% RSLogix 500 project Planer 3-1-07.RSS, saved by version 7.00.00.19 %
PROJECT "PLANER"    % processor: MicroLogix 1500 %

PROGRAM FILES
  LAD 2 "MAIN"  13 rungs
  LAD 3 "INFEED"  10 rungs
  LAD 4 "TILTHOIST"  9 rungs
  LAD 5 "GRADING"  22 rungs
  LAD 6 "PLANER IF"  6 rungs
  LAD 7 "PLANER OF"  5 rungs
  LAD 8 "MR CONVS"  7 rungs
  LAD 9 "CYCLONE"  3 rungs
  LAD 10 "INDICATION"  11 rungs

DATA FILES
  O0 OUTPUT  9 elements
  I1 INPUT  8 elements
  S2 STATUS  66 elements
  B3 BINARY  10 elements
  T4 TIMER  34 elements
  C5 COUNTER  1 elements
  R6 CONTROL  1 elements
  N7 INTEGER  1 elements
  F8 FLOAT  1 elements

LADDER 2 "MAIN"
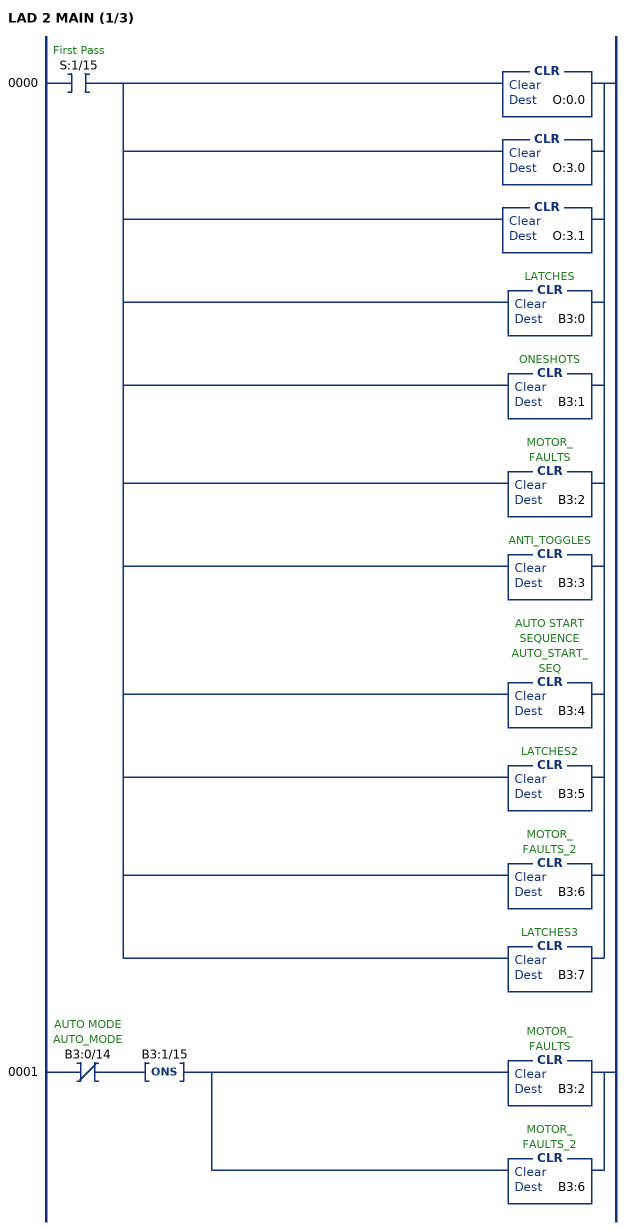
% Rung: 0 %
SOR XIC S:1/15 BST CLR O:0.0 NXB CLR O:3.0 NXB CLR O:3.1 NXB CLR B3:0 NXB CLR B3:1 NXB CLR B3:2 NXB CLR B3:3 NXB CLR B3:4 NXB CLR B3:5 NXB CLR B3:6 NXB CLR B3:7 BND EOR
%   S:1/15  "First Pass" %
%   B3:0  LATCHES %
%   B3:1  ONESHOTS %
%   B3:2  MOTOR_FAULTS %
%   B3:3  ANTI_TOGGLES %
%   B3:4  AUTO_START_SEQ  "AUTO START SEQUENCE" %
%   B3:5  LATCHES2 %
%   B3:6  MOTOR_FAULTS_2 %
%   B3:7  LATCHES3 %
% Rung: 1 %
SOR XIO B3:0/14 ONS B3:1/15 BST CLR B3:2 NXB CLR B3:6 BND EOR
%   B3:0/14  AUTO_MODE  "AUTO MODE" %
%   B3:2  MOTOR_FAULTS %
%   B3:6  MOTOR_FAULTS_2 %

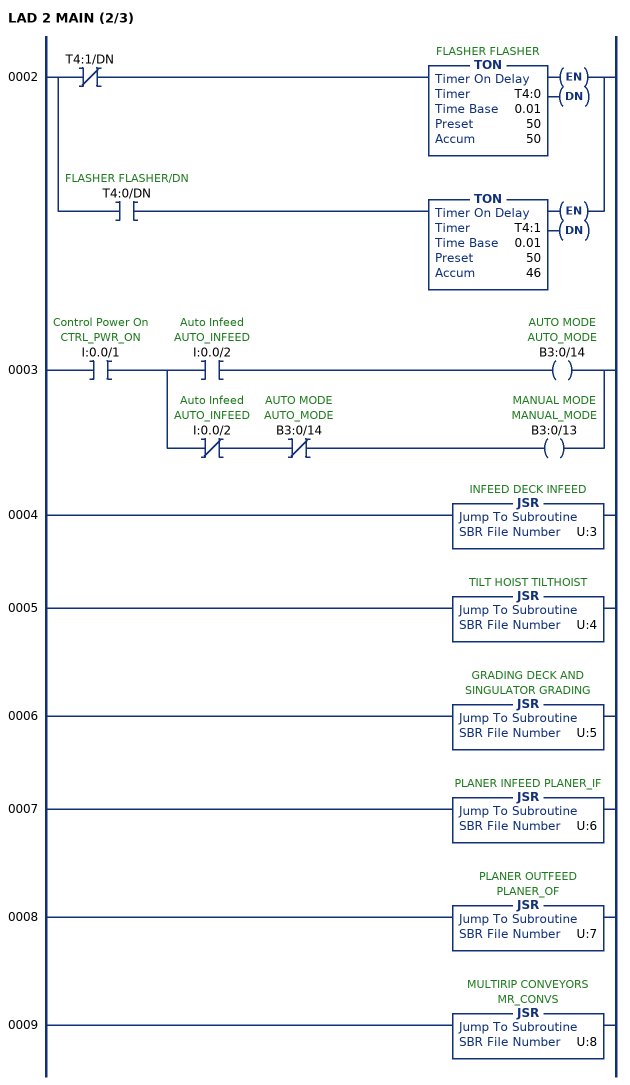
% Rung: 2 %
SOR BST XIO T4:1/DN TON T4:0 0.01 50 50 NXB XIC T4:0/DN TON T4:1 0.01 50 46 BND EOR
%   T4:0  FLASHER  "FLASHER" %
% Rung: 3 %
SOR XIC I:0.0/1 BST XIC I:0.0/2 OTE B3:0/14 NXB XIO I:0.0/2 XIO B3:0/14 OTE B3:0/13 BND EOR
%   I:0.0/1  CTRL_PWR_ON  "Control Power On" %
%   I:0.0/2  AUTO_INFEED  "Auto Infeed" %
%   B3:0/14  AUTO_MODE  "AUTO MODE" %
%   B3:0/13  MANUAL_MODE  "MANUAL MODE" %
% Rung: 4 %
SOR JSR U:3 EOR
%   U:3  INFEED  "INFEED DECK" %
% Rung: 5 %
SOR JSR U:4 EOR
%   U:4  TILTHOIST  "TILT HOIST" %
% Rung: 6 %
SOR JSR U:5 EOR
%   U:5  GRADING  "GRADING DECK AND SINGULATOR" %
% Rung: 7 %
SOR JSR U:6 EOR
%   U:6  PLANER_IF  "PLANER INFEED" %
% Rung: 8 %
SOR JSR U:7 EOR
%   U:7  PLANER_OF  "PLANER OUTFEED" %
% Rung: 9 %
SOR JSR U:8 EOR
%   U:8  MR_CONVS  "MULTIRIP CONVEYORS" %

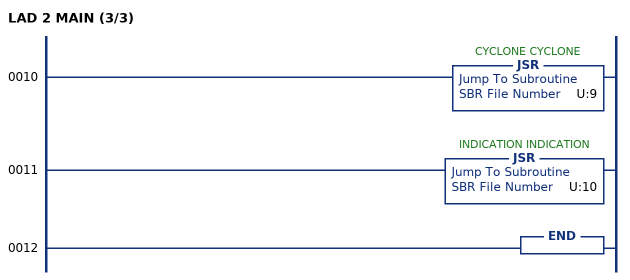
% Rung: 10 %
SOR JSR U:9 EOR
%   U:9  CYCLONE  "CYCLONE" %
% Rung: 11 %
SOR JSR U:10 EOR
%   U:10  INDICATION  "INDICATION" %
% Rung: 12 %
SOR END EOR

LADDER 3 "INFEED"
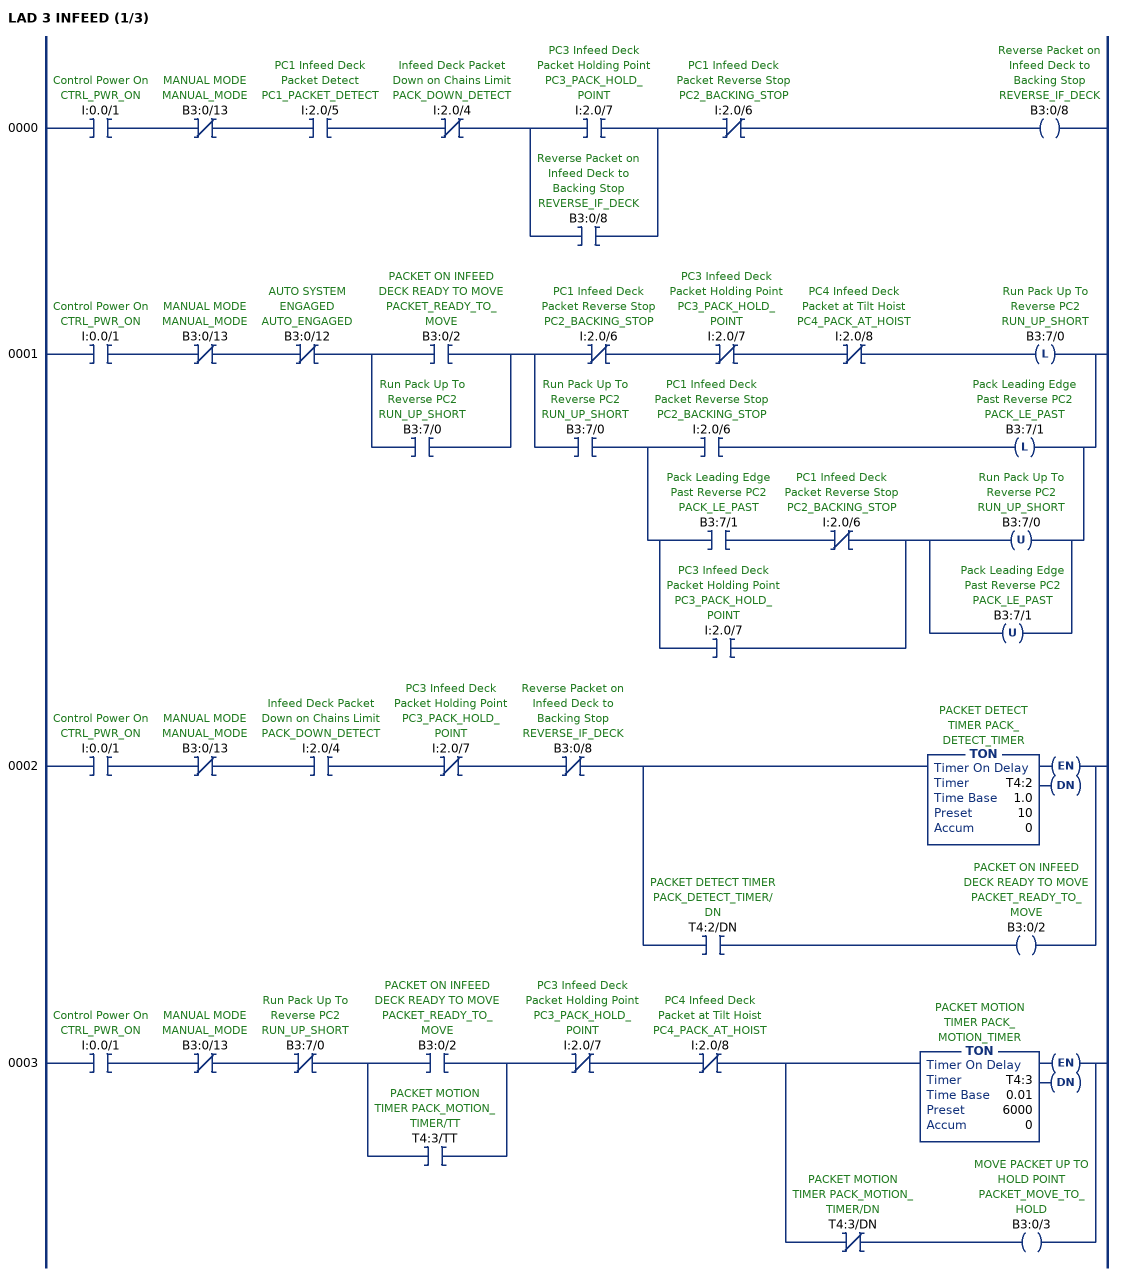
% Rung: 0 %
SOR XIC I:0.0/1 XIO B3:0/13 XIC I:2.0/5 XIO I:2.0/4 BST XIC I:2.0/7 NXB XIC B3:0/8 BND XIO I:2.0/6 OTE B3:0/8 EOR
%   I:0.0/1  CTRL_PWR_ON  "Control Power On" %
%   B3:0/13  MANUAL_MODE  "MANUAL MODE" %
%   I:2.0/5  PC1_PACKET_DETECT  "PC1 Infeed Deck Packet Detect" %
%   I:2.0/4  PACK_DOWN_DETECT  "Infeed Deck Packet Down on Chains Limit" %
%   I:2.0/7  PC3_PACK_HOLD_POINT  "PC3 Infeed Deck Packet Holding Point" %
%   B3:0/8  REVERSE_IF_DECK  "Reverse Packet on Infeed Deck to Backing Stop" %
%   I:2.0/6  PC2_BACKING_STOP  "PC1 Infeed Deck Packet Reverse Stop" %
% Rung: 1 %
SOR XIC I:0.0/1 XIO B3:0/13 XIO B3:0/12 BST XIC B3:0/2 NXB XIC B3:7/0 BND BST XIO I:2.0/6 XIO I:2.0/7 XIO I:2.0/8 OTL B3:7/0 NXB XIC B3:7/0 BST XIC I:2.0/6 OTL B3:7/1 NXB BST XIC B3:7/1 XIO I:2.0/6 NXB XIC I:2.0/7 BND BST OTU B3:7/0 NXB OTU B3:7/1 BND BND BND EOR
%   I:0.0/1  CTRL_PWR_ON  "Control Power On" %
%   B3:0/13  MANUAL_MODE  "MANUAL MODE" %
%   B3:0/12  AUTO_ENGAGED  "AUTO SYSTEM ENGAGED" %
%   B3:0/2  PACKET_READY_TO_MOVE  "PACKET ON INFEED DECK READY TO MOVE" %
%   B3:7/0  RUN_UP_SHORT  "Run Pack Up To Reverse PC2" %
%   I:2.0/6  PC2_BACKING_STOP  "PC1 Infeed Deck Packet Reverse Stop" %
%   I:2.0/7  PC3_PACK_HOLD_POINT  "PC3 Infeed Deck Packet Holding Point" %
%   I:2.0/8  PC4_PACK_AT_HOIST  "PC4 Infeed Deck Packet at Tilt Hoist" %
%   B3:7/1  PACK_LE_PAST  "Pack Leading Edge Past Reverse PC2" %
% Rung: 2 %
SOR XIC I:0.0/1 XIO B3:0/13 XIC I:2.0/4 XIO I:2.0/7 XIO B3:0/8 BST TON T4:2 1.0 10 0 NXB XIC T4:2/DN OTE B3:0/2 BND EOR
%   I:0.0/1  CTRL_PWR_ON  "Control Power On" %
%   B3:0/13  MANUAL_MODE  "MANUAL MODE" %
%   I:2.0/4  PACK_DOWN_DETECT  "Infeed Deck Packet Down on Chains Limit" %
%   I:2.0/7  PC3_PACK_HOLD_POINT  "PC3 Infeed Deck Packet Holding Point" %
%   B3:0/8  REVERSE_IF_DECK  "Reverse Packet on Infeed Deck to Backing Stop" %
%   T4:2  PACK_DETECT_TIMER  "PACKET DETECT TIMER" %
%   B3:0/2  PACKET_READY_TO_MOVE  "PACKET ON INFEED DECK READY TO MOVE" %
% Rung: 3 %
SOR XIC I:0.0/1 XIO B3:0/13 XIO B3:7/0 BST XIC B3:0/2 NXB XIC T4:3/TT BND XIO I:2.0/7 XIO I:2.0/8 BST TON T4:3 0.01 6000 0 NXB XIO T4:3/DN OTE B3:0/3 BND EOR
%   I:0.0/1  CTRL_PWR_ON  "Control Power On" %
%   B3:0/13  MANUAL_MODE  "MANUAL MODE" %
%   B3:7/0  RUN_UP_SHORT  "Run Pack Up To Reverse PC2" %
%   B3:0/2  PACKET_READY_TO_MOVE  "PACKET ON INFEED DECK READY TO MOVE" %
%   T4:3  PACK_MOTION_TIMER  "PACKET MOTION TIMER" %
%   I:2.0/7  PC3_PACK_HOLD_POINT  "PC3 Infeed Deck Packet Holding Point" %
%   I:2.0/8  PC4_PACK_AT_HOIST  "PC4 Infeed Deck Packet at Tilt Hoist" %
%   B3:0/3  PACKET_MOVE_TO_HOLD  "MOVE PACKET UP TO HOLD POINT" %

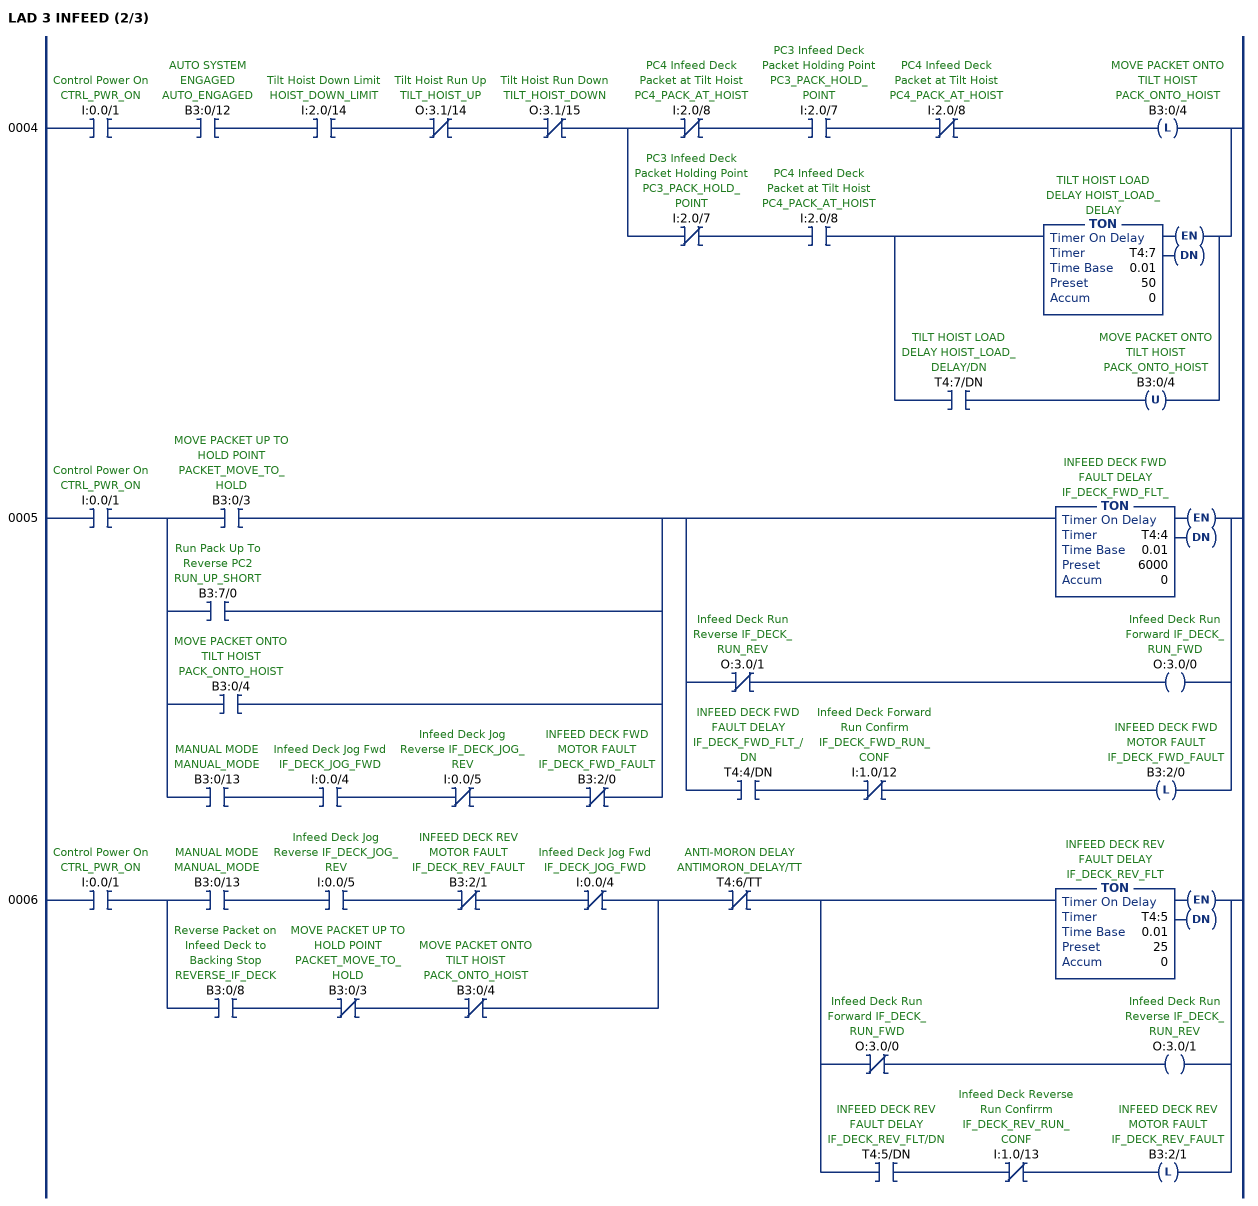
% Rung: 4 %
SOR XIC I:0.0/1 XIC B3:0/12 XIC I:2.0/14 XIO O:3.1/14 XIO O:3.1/15 BST XIO I:2.0/8 XIC I:2.0/7 XIO I:2.0/8 OTL B3:0/4 NXB XIO I:2.0/7 XIC I:2.0/8 BST TON T4:7 0.01 50 0 NXB XIC T4:7/DN OTU B3:0/4 BND BND EOR
%   I:0.0/1  CTRL_PWR_ON  "Control Power On" %
%   B3:0/12  AUTO_ENGAGED  "AUTO SYSTEM ENGAGED" %
%   I:2.0/14  HOIST_DOWN_LIMIT  "Tilt Hoist Down Limit" %
%   O:3.1/14  TILT_HOIST_UP  "Tilt Hoist Run Up" %
%   O:3.1/15  TILT_HOIST_DOWN  "Tilt Hoist Run Down" %
%   I:2.0/8  PC4_PACK_AT_HOIST  "PC4 Infeed Deck Packet at Tilt Hoist" %
%   I:2.0/7  PC3_PACK_HOLD_POINT  "PC3 Infeed Deck Packet Holding Point" %
%   B3:0/4  PACK_ONTO_HOIST  "MOVE PACKET ONTO TILT HOIST" %
%   T4:7  HOIST_LOAD_DELAY  "TILT HOIST LOAD DELAY" %
% Rung: 5 %
SOR XIC I:0.0/1 BST BST XIC B3:0/3 NXB XIC B3:7/0 NXB XIC B3:0/4 BND NXB XIC B3:0/13 XIC I:0.0/4 XIO I:0.0/5 XIO B3:2/0 BND BST TON T4:4 0.01 6000 0 NXB XIO O:3.0/1 OTE O:3.0/0 NXB XIC T4:4/DN XIO I:1.0/12 OTL B3:2/0 BND EOR
%   I:0.0/1  CTRL_PWR_ON  "Control Power On" %
%   B3:0/3  PACKET_MOVE_TO_HOLD  "MOVE PACKET UP TO HOLD POINT" %
%   B3:7/0  RUN_UP_SHORT  "Run Pack Up To Reverse PC2" %
%   B3:0/4  PACK_ONTO_HOIST  "MOVE PACKET ONTO TILT HOIST" %
%   B3:0/13  MANUAL_MODE  "MANUAL MODE" %
%   I:0.0/4  IF_DECK_JOG_FWD  "Infeed Deck Jog Fwd" %
%   I:0.0/5  IF_DECK_JOG_REV  "Infeed Deck Jog Reverse" %
%   B3:2/0  IF_DECK_FWD_FAULT  "INFEED DECK FWD MOTOR FAULT" %
%   T4:4  IF_DECK_FWD_FLT_  "INFEED DECK FWD FAULT DELAY" %
%   O:3.0/1  IF_DECK_RUN_REV  "Infeed Deck Run Reverse" %
%   O:3.0/0  IF_DECK_RUN_FWD  "Infeed Deck Run Forward" %
%   I:1.0/12  IF_DECK_FWD_RUN_CONF  "Infeed Deck Forward Run Confirm" %
% Rung: 6 %
SOR XIC I:0.0/1 BST XIC B3:0/13 XIC I:0.0/5 XIO B3:2/1 XIO I:0.0/4 NXB XIC B3:0/8 XIO B3:0/3 XIO B3:0/4 BND XIO T4:6/TT BST TON T4:5 0.01 25 0 NXB XIO O:3.0/0 OTE O:3.0/1 NXB XIC T4:5/DN XIO I:1.0/13 OTL B3:2/1 BND EOR
%   I:0.0/1  CTRL_PWR_ON  "Control Power On" %
%   B3:0/13  MANUAL_MODE  "MANUAL MODE" %
%   I:0.0/5  IF_DECK_JOG_REV  "Infeed Deck Jog Reverse" %
%   B3:2/1  IF_DECK_REV_FAULT  "INFEED DECK REV MOTOR FAULT" %
%   I:0.0/4  IF_DECK_JOG_FWD  "Infeed Deck Jog Fwd" %
%   B3:0/8  REVERSE_IF_DECK  "Reverse Packet on Infeed Deck to Backing Stop" %
%   B3:0/3  PACKET_MOVE_TO_HOLD  "MOVE PACKET UP TO HOLD POINT" %
%   B3:0/4  PACK_ONTO_HOIST  "MOVE PACKET ONTO TILT HOIST" %
%   T4:6  ANTIMORON_DELAY  "ANTI-MORON DELAY" %
%   T4:5  IF_DECK_REV_FLT  "INFEED DECK REV FAULT DELAY" %
%   O:3.0/0  IF_DECK_RUN_FWD  "Infeed Deck Run Forward" %
%   O:3.0/1  IF_DECK_RUN_REV  "Infeed Deck Run Reverse" %
%   I:1.0/13  IF_DECK_REV_RUN_CONF  "Infeed Deck Reverse Run Confirrm" %

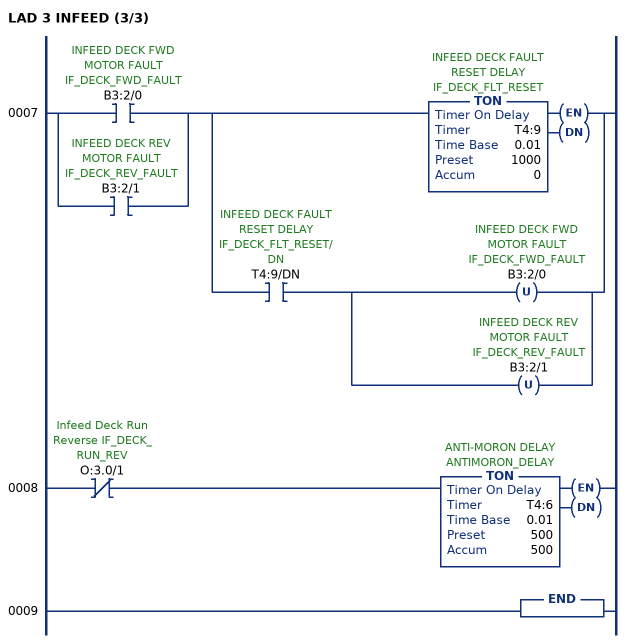
% Rung: 7 %
SOR BST XIC B3:2/0 NXB XIC B3:2/1 BND BST TON T4:9 0.01 1000 0 NXB XIC T4:9/DN BST OTU B3:2/0 NXB OTU B3:2/1 BND BND EOR
%   B3:2/0  IF_DECK_FWD_FAULT  "INFEED DECK FWD MOTOR FAULT" %
%   B3:2/1  IF_DECK_REV_FAULT  "INFEED DECK REV MOTOR FAULT" %
%   T4:9  IF_DECK_FLT_RESET  "INFEED DECK FAULT RESET DELAY" %
% Rung: 8 %
SOR XIO O:3.0/1 TON T4:6 0.01 500 500 EOR
%   O:3.0/1  IF_DECK_RUN_REV  "Infeed Deck Run Reverse" %
%   T4:6  ANTIMORON_DELAY  "ANTI-MORON DELAY" %
% Rung: 9 %
SOR END EOR

LADDER 4 "TILTHOIST"
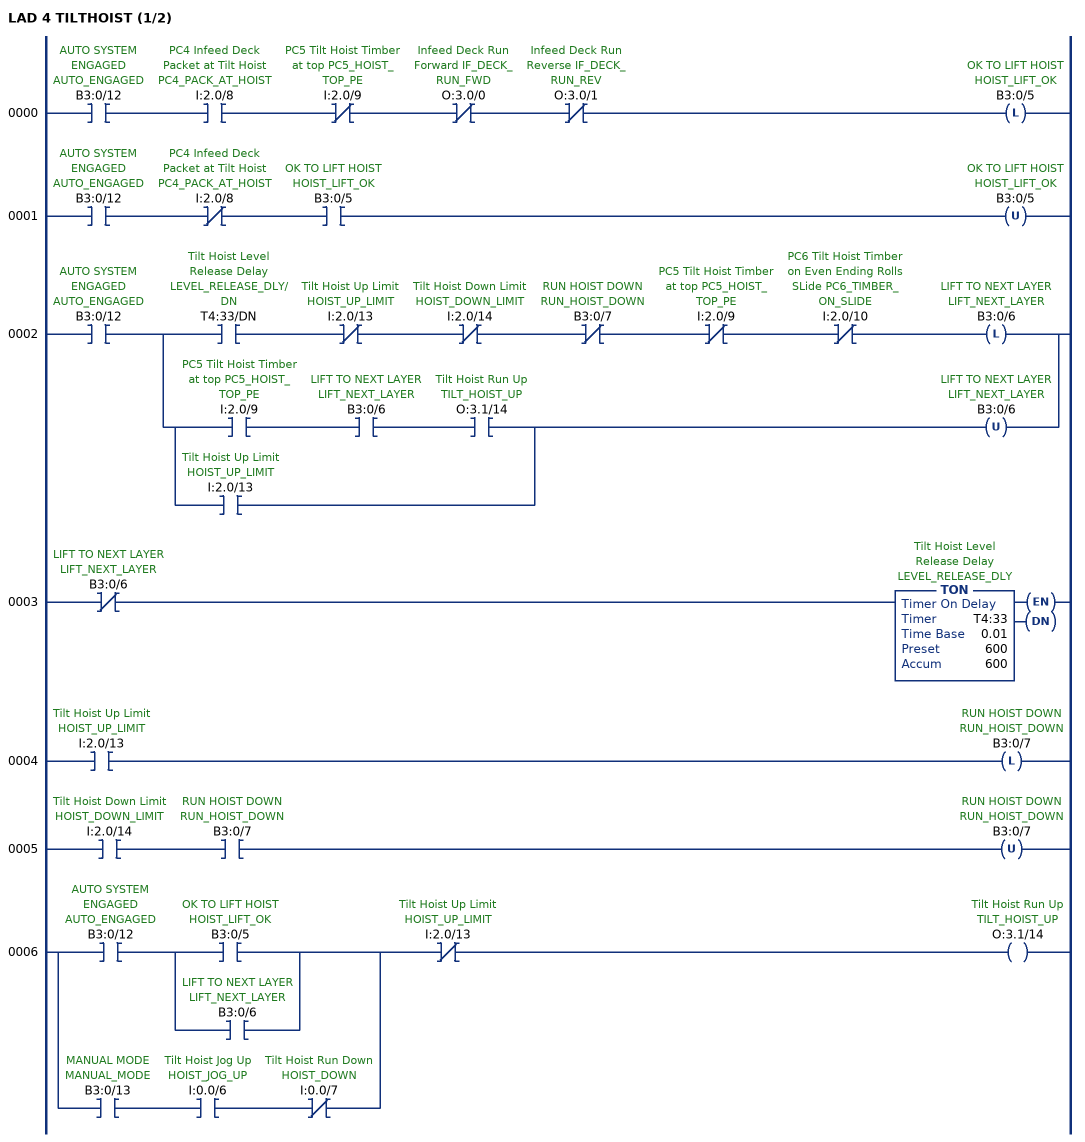
% Rung: 0 %
SOR XIC B3:0/12 XIC I:2.0/8 XIO I:2.0/9 XIO O:3.0/0 XIO O:3.0/1 OTL B3:0/5 EOR
%   B3:0/12  AUTO_ENGAGED  "AUTO SYSTEM ENGAGED" %
%   I:2.0/8  PC4_PACK_AT_HOIST  "PC4 Infeed Deck Packet at Tilt Hoist" %
%   I:2.0/9  PC5_HOIST_TOP_PE  "PC5 Tilt Hoist Timber at top" %
%   O:3.0/0  IF_DECK_RUN_FWD  "Infeed Deck Run Forward" %
%   O:3.0/1  IF_DECK_RUN_REV  "Infeed Deck Run Reverse" %
%   B3:0/5  HOIST_LIFT_OK  "OK TO LIFT HOIST" %
% Rung: 1 %
SOR XIC B3:0/12 XIO I:2.0/8 XIC B3:0/5 OTU B3:0/5 EOR
%   B3:0/12  AUTO_ENGAGED  "AUTO SYSTEM ENGAGED" %
%   I:2.0/8  PC4_PACK_AT_HOIST  "PC4 Infeed Deck Packet at Tilt Hoist" %
%   B3:0/5  HOIST_LIFT_OK  "OK TO LIFT HOIST" %
% Rung: 2 %
SOR XIC B3:0/12 BST XIC T4:33/DN XIO I:2.0/13 XIO I:2.0/14 XIO B3:0/7 XIO I:2.0/9 XIO I:2.0/10 OTL B3:0/6 NXB BST XIC I:2.0/9 XIC B3:0/6 XIC O:3.1/14 NXB XIC I:2.0/13 BND OTU B3:0/6 BND EOR
%   B3:0/12  AUTO_ENGAGED  "AUTO SYSTEM ENGAGED" %
%   T4:33  LEVEL_RELEASE_DLY  "Tilt Hoist Level Release Delay" %
%   I:2.0/13  HOIST_UP_LIMIT  "Tilt Hoist Up Limit" %
%   I:2.0/14  HOIST_DOWN_LIMIT  "Tilt Hoist Down Limit" %
%   B3:0/7  RUN_HOIST_DOWN  "RUN HOIST DOWN" %
%   I:2.0/9  PC5_HOIST_TOP_PE  "PC5 Tilt Hoist Timber at top" %
%   I:2.0/10  PC6_TIMBER_ON_SLIDE  "PC6 Tilt Hoist Timber on Even Ending Rolls SLide" %
%   B3:0/6  LIFT_NEXT_LAYER  "LIFT TO NEXT LAYER" %
%   O:3.1/14  TILT_HOIST_UP  "Tilt Hoist Run Up" %
% Rung: 3 %
SOR XIO B3:0/6 TON T4:33 0.01 600 600 EOR
%   B3:0/6  LIFT_NEXT_LAYER  "LIFT TO NEXT LAYER" %
%   T4:33  LEVEL_RELEASE_DLY  "Tilt Hoist Level Release Delay" %
% Rung: 4 %
SOR XIC I:2.0/13 OTL B3:0/7 EOR
%   I:2.0/13  HOIST_UP_LIMIT  "Tilt Hoist Up Limit" %
%   B3:0/7  RUN_HOIST_DOWN  "RUN HOIST DOWN" %
% Rung: 5 %
SOR XIC I:2.0/14 XIC B3:0/7 OTU B3:0/7 EOR
%   I:2.0/14  HOIST_DOWN_LIMIT  "Tilt Hoist Down Limit" %
%   B3:0/7  RUN_HOIST_DOWN  "RUN HOIST DOWN" %
% Rung: 6 %
SOR BST XIC B3:0/12 BST XIC B3:0/5 NXB XIC B3:0/6 BND NXB XIC B3:0/13 XIC I:0.0/6 XIO I:0.0/7 BND XIO I:2.0/13 OTE O:3.1/14 EOR
%   B3:0/12  AUTO_ENGAGED  "AUTO SYSTEM ENGAGED" %
%   B3:0/5  HOIST_LIFT_OK  "OK TO LIFT HOIST" %
%   B3:0/6  LIFT_NEXT_LAYER  "LIFT TO NEXT LAYER" %
%   B3:0/13  MANUAL_MODE  "MANUAL MODE" %
%   I:0.0/6  HOIST_JOG_UP  "Tilt Hoist Jog Up" %
%   I:0.0/7  HOIST_DOWN  "Tilt Hoist Run Down" %
%   I:2.0/13  HOIST_UP_LIMIT  "Tilt Hoist Up Limit" %
%   O:3.1/14  TILT_HOIST_UP  "Tilt Hoist Run Up" %

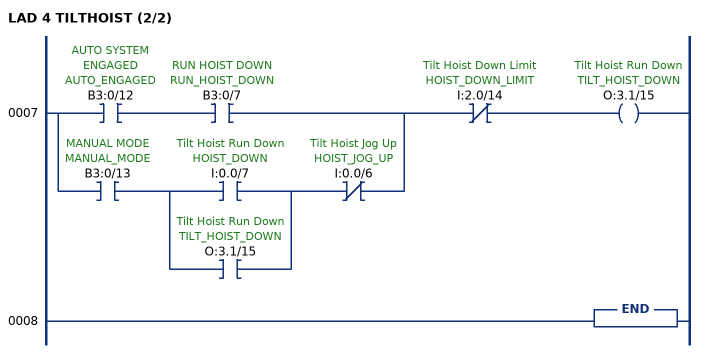
% Rung: 7 %
SOR BST XIC B3:0/12 XIC B3:0/7 NXB XIC B3:0/13 BST XIC I:0.0/7 NXB XIC O:3.1/15 BND XIO I:0.0/6 BND XIO I:2.0/14 OTE O:3.1/15 EOR
%   B3:0/12  AUTO_ENGAGED  "AUTO SYSTEM ENGAGED" %
%   B3:0/7  RUN_HOIST_DOWN  "RUN HOIST DOWN" %
%   B3:0/13  MANUAL_MODE  "MANUAL MODE" %
%   I:0.0/7  HOIST_DOWN  "Tilt Hoist Run Down" %
%   O:3.1/15  TILT_HOIST_DOWN  "Tilt Hoist Run Down" %
%   I:0.0/6  HOIST_JOG_UP  "Tilt Hoist Jog Up" %
%   I:2.0/14  HOIST_DOWN_LIMIT  "Tilt Hoist Down Limit" %
% Rung: 8 %
SOR END EOR

LADDER 5 "GRADING"
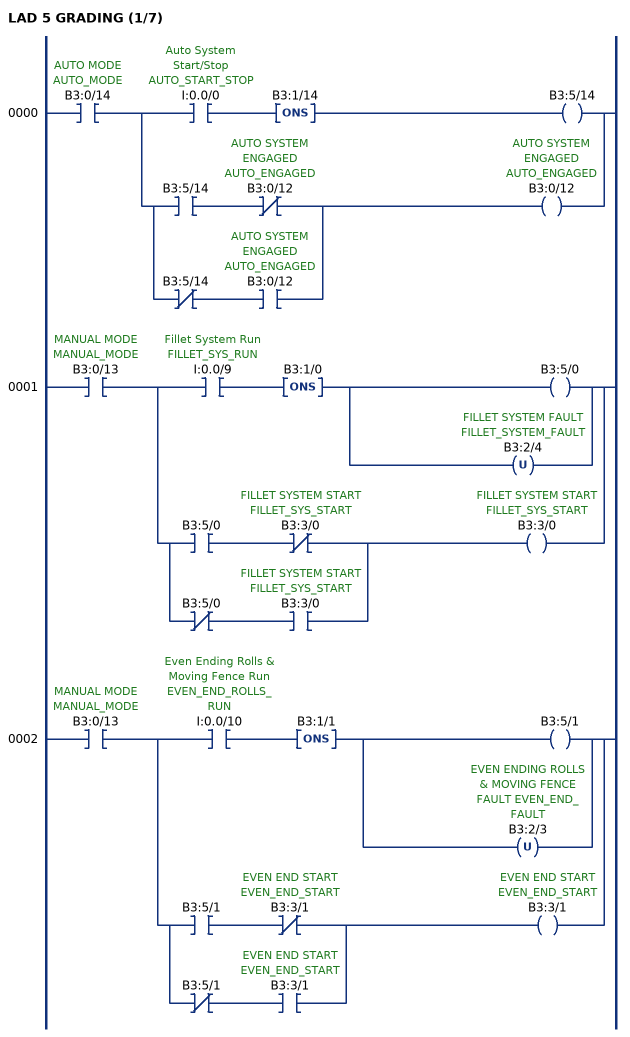
% Rung: 0 %
SOR XIC B3:0/14 BST XIC I:0.0/0 ONS B3:1/14 OTE B3:5/14 NXB BST XIC B3:5/14 XIO B3:0/12 NXB XIO B3:5/14 XIC B3:0/12 BND OTE B3:0/12 BND EOR
%   B3:0/14  AUTO_MODE  "AUTO MODE" %
%   I:0.0/0  AUTO_START_STOP  "Auto System Start/Stop" %
%   B3:0/12  AUTO_ENGAGED  "AUTO SYSTEM ENGAGED" %
% Rung: 1 %
SOR XIC B3:0/13 BST XIC I:0.0/9 ONS B3:1/0 BST OTE B3:5/0 NXB OTU B3:2/4 BND NXB BST XIC B3:5/0 XIO B3:3/0 NXB XIO B3:5/0 XIC B3:3/0 BND OTE B3:3/0 BND EOR
%   B3:0/13  MANUAL_MODE  "MANUAL MODE" %
%   I:0.0/9  FILLET_SYS_RUN  "Fillet System Run" %
%   B3:2/4  FILLET_SYSTEM_FAULT  "FILLET SYSTEM FAULT" %
%   B3:3/0  FILLET_SYS_START  "FILLET SYSTEM START" %
% Rung: 2 %
SOR XIC B3:0/13 BST XIC I:0.0/10 ONS B3:1/1 BST OTE B3:5/1 NXB OTU B3:2/3 BND NXB BST XIC B3:5/1 XIO B3:3/1 NXB XIO B3:5/1 XIC B3:3/1 BND OTE B3:3/1 BND EOR
%   B3:0/13  MANUAL_MODE  "MANUAL MODE" %
%   I:0.0/10  EVEN_END_ROLLS_RUN  "Even Ending Rolls & Moving Fence Run" %
%   B3:2/3  EVEN_END_FAULT  "EVEN ENDING ROLLS & MOVING FENCE FAULT" %
%   B3:3/1  EVEN_END_START  "EVEN END START" %

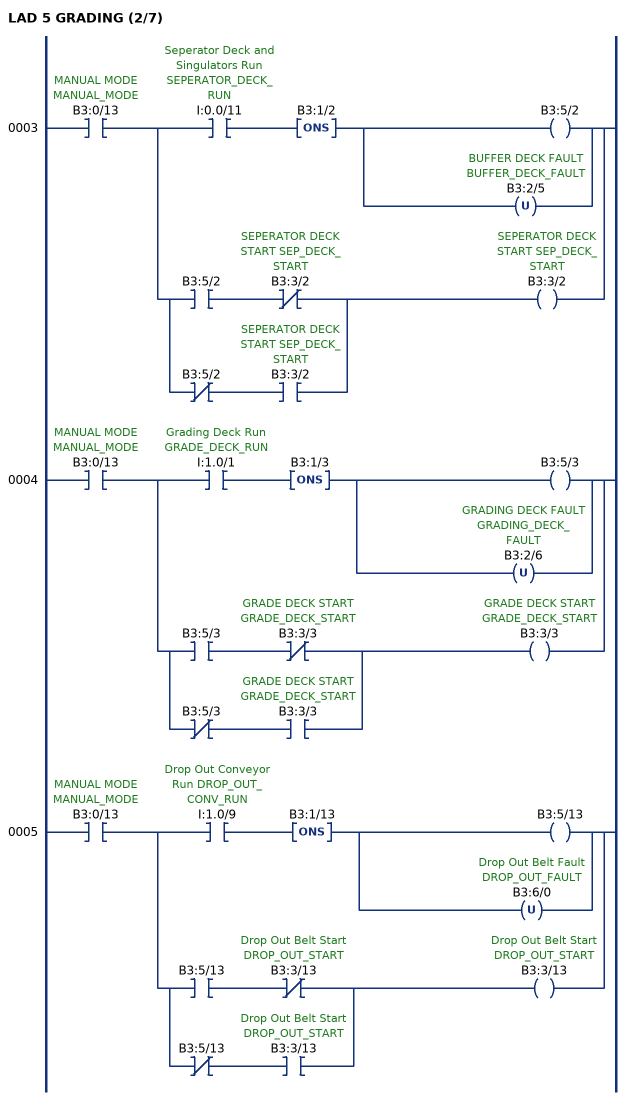
% Rung: 3 %
SOR XIC B3:0/13 BST XIC I:0.0/11 ONS B3:1/2 BST OTE B3:5/2 NXB OTU B3:2/5 BND NXB BST XIC B3:5/2 XIO B3:3/2 NXB XIO B3:5/2 XIC B3:3/2 BND OTE B3:3/2 BND EOR
%   B3:0/13  MANUAL_MODE  "MANUAL MODE" %
%   I:0.0/11  SEPERATOR_DECK_RUN  "Seperator Deck and Singulators Run" %
%   B3:2/5  BUFFER_DECK_FAULT  "BUFFER DECK FAULT" %
%   B3:3/2  SEP_DECK_START  "SEPERATOR DECK START" %
% Rung: 4 %
SOR XIC B3:0/13 BST XIC I:1.0/1 ONS B3:1/3 BST OTE B3:5/3 NXB OTU B3:2/6 BND NXB BST XIC B3:5/3 XIO B3:3/3 NXB XIO B3:5/3 XIC B3:3/3 BND OTE B3:3/3 BND EOR
%   B3:0/13  MANUAL_MODE  "MANUAL MODE" %
%   I:1.0/1  GRADE_DECK_RUN  "Grading Deck Run" %
%   B3:2/6  GRADING_DECK_FAULT  "GRADING DECK FAULT" %
%   B3:3/3  GRADE_DECK_START  "GRADE DECK START" %
% Rung: 5 %
SOR XIC B3:0/13 BST XIC I:1.0/9 ONS B3:1/13 BST OTE B3:5/13 NXB OTU B3:6/0 BND NXB BST XIC B3:5/13 XIO B3:3/13 NXB XIO B3:5/13 XIC B3:3/13 BND OTE B3:3/13 BND EOR
%   B3:0/13  MANUAL_MODE  "MANUAL MODE" %
%   I:1.0/9  DROP_OUT_CONV_RUN  "Drop Out Conveyor Run" %
%   B3:6/0  DROP_OUT_FAULT  "Drop Out Belt Fault" %
%   B3:3/13  DROP_OUT_START  "Drop Out Belt Start" %

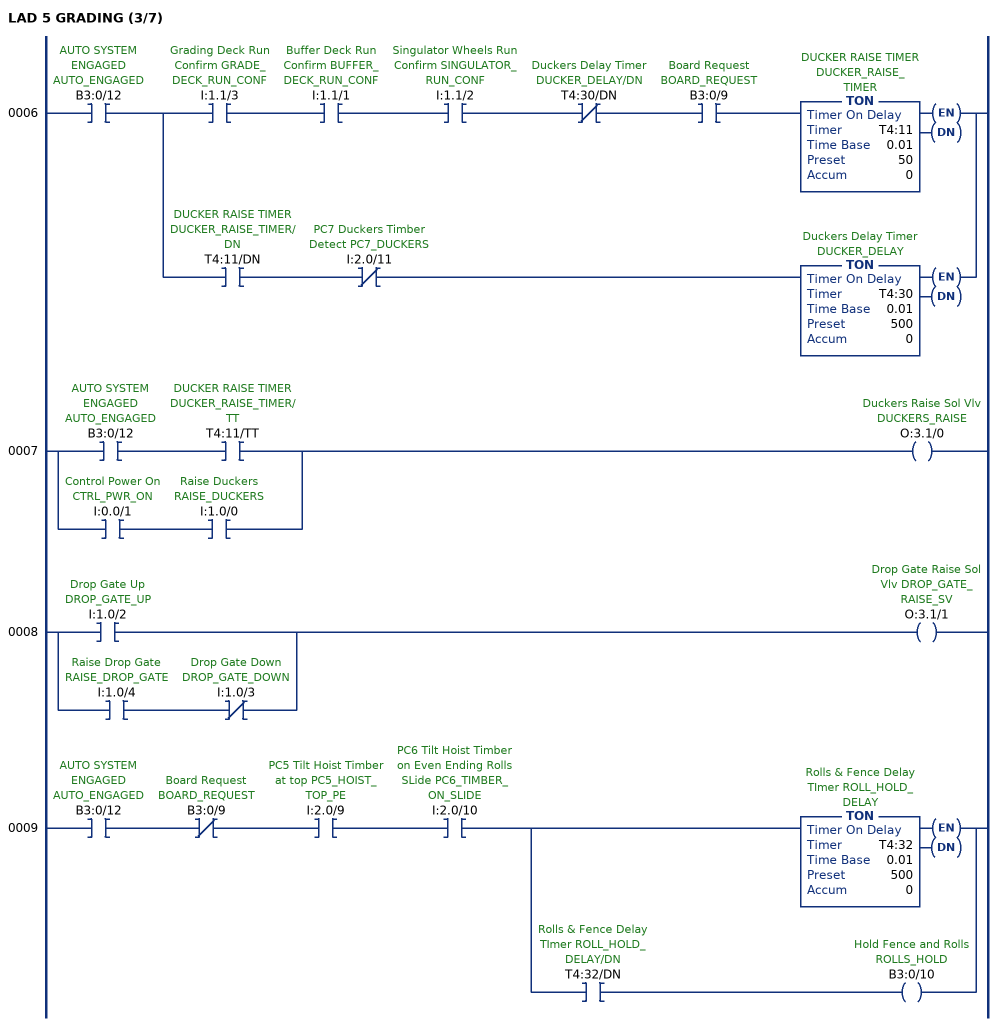
% Rung: 6 %
SOR XIC B3:0/12 BST XIC I:1.1/3 XIC I:1.1/1 XIC I:1.1/2 XIO T4:30/DN XIC B3:0/9 TON T4:11 0.01 50 0 NXB XIC T4:11/DN XIO I:2.0/11 TON T4:30 0.01 500 0 BND EOR
%   B3:0/12  AUTO_ENGAGED  "AUTO SYSTEM ENGAGED" %
%   I:1.1/3  GRADE_DECK_RUN_CONF  "Grading Deck Run Confirm" %
%   I:1.1/1  BUFFER_DECK_RUN_CONF  "Buffer Deck Run Confirm" %
%   I:1.1/2  SINGULATOR_RUN_CONF  "Singulator Wheels Run Confirm" %
%   T4:30  DUCKER_DELAY  "Duckers Delay Timer" %
%   B3:0/9  BOARD_REQUEST  "Board Request" %
%   T4:11  DUCKER_RAISE_TIMER  "DUCKER RAISE TIMER" %
%   I:2.0/11  PC7_DUCKERS  "PC7 Duckers Timber Detect" %
% Rung: 7 %
SOR BST XIC B3:0/12 XIC T4:11/TT NXB XIC I:0.0/1 XIC I:1.0/0 BND OTE O:3.1/0 EOR
%   B3:0/12  AUTO_ENGAGED  "AUTO SYSTEM ENGAGED" %
%   T4:11  DUCKER_RAISE_TIMER  "DUCKER RAISE TIMER" %
%   I:0.0/1  CTRL_PWR_ON  "Control Power On" %
%   I:1.0/0  RAISE_DUCKERS  "Raise Duckers" %
%   O:3.1/0  DUCKERS_RAISE  "Duckers Raise Sol Vlv" %
% Rung: 8 %
SOR BST XIC I:1.0/2 NXB XIC I:1.0/4 XIO I:1.0/3 BND OTE O:3.1/1 EOR
%   I:1.0/2  DROP_GATE_UP  "Drop Gate Up" %
%   I:1.0/4  RAISE_DROP_GATE  "Raise Drop Gate" %
%   I:1.0/3  DROP_GATE_DOWN  "Drop Gate Down" %
%   O:3.1/1  DROP_GATE_RAISE_SV  "Drop Gate Raise Sol Vlv" %
% Rung: 9 %
SOR XIC B3:0/12 XIO B3:0/9 XIC I:2.0/9 XIC I:2.0/10 BST TON T4:32 0.01 500 0 NXB XIC T4:32/DN OTE B3:0/10 BND EOR
%   B3:0/12  AUTO_ENGAGED  "AUTO SYSTEM ENGAGED" %
%   B3:0/9  BOARD_REQUEST  "Board Request" %
%   I:2.0/9  PC5_HOIST_TOP_PE  "PC5 Tilt Hoist Timber at top" %
%   I:2.0/10  PC6_TIMBER_ON_SLIDE  "PC6 Tilt Hoist Timber on Even Ending Rolls SLide" %
%   T4:32  ROLL_HOLD_DELAY  "Rolls & Fence Delay TImer" %
%   B3:0/10  ROLLS_HOLD  "Hold Fence and Rolls" %

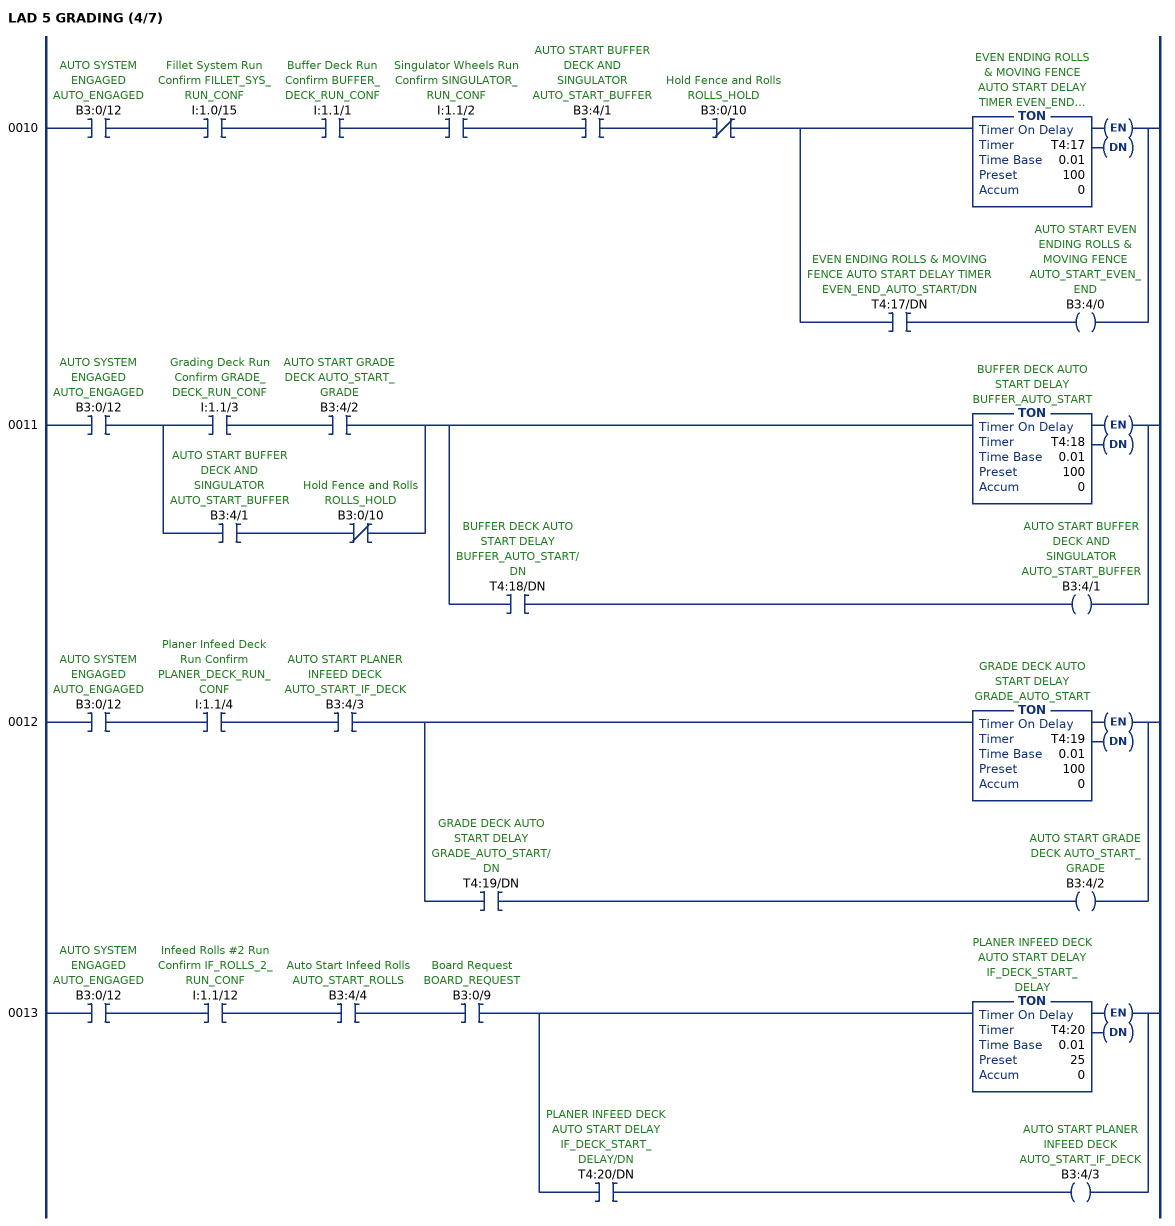
% Rung: 10 %
SOR XIC B3:0/12 XIC I:1.0/15 XIC I:1.1/1 XIC I:1.1/2 XIC B3:4/1 XIO B3:0/10 BST TON T4:17 0.01 100 0 NXB XIC T4:17/DN OTE B3:4/0 BND EOR
%   B3:0/12  AUTO_ENGAGED  "AUTO SYSTEM ENGAGED" %
%   I:1.0/15  FILLET_SYS_RUN_CONF  "Fillet System Run Confirm" %
%   I:1.1/1  BUFFER_DECK_RUN_CONF  "Buffer Deck Run Confirm" %
%   I:1.1/2  SINGULATOR_RUN_CONF  "Singulator Wheels Run Confirm" %
%   B3:4/1  AUTO_START_BUFFER  "AUTO START BUFFER DECK AND SINGULATOR" %
%   B3:0/10  ROLLS_HOLD  "Hold Fence and Rolls" %
%   T4:17  EVEN_END_AUTO_START  "EVEN ENDING ROLLS & MOVING FENCE AUTO START DELAY TIMER" %
%   B3:4/0  AUTO_START_EVEN_END  "AUTO START EVEN ENDING ROLLS & MOVING FENCE" %
% Rung: 11 %
SOR XIC B3:0/12 BST XIC I:1.1/3 XIC B3:4/2 NXB XIC B3:4/1 XIO B3:0/10 BND BST TON T4:18 0.01 100 0 NXB XIC T4:18/DN OTE B3:4/1 BND EOR
%   B3:0/12  AUTO_ENGAGED  "AUTO SYSTEM ENGAGED" %
%   I:1.1/3  GRADE_DECK_RUN_CONF  "Grading Deck Run Confirm" %
%   B3:4/2  AUTO_START_GRADE  "AUTO START GRADE DECK" %
%   B3:4/1  AUTO_START_BUFFER  "AUTO START BUFFER DECK AND SINGULATOR" %
%   B3:0/10  ROLLS_HOLD  "Hold Fence and Rolls" %
%   T4:18  BUFFER_AUTO_START  "BUFFER DECK AUTO START DELAY" %
% Rung: 12 %
SOR XIC B3:0/12 XIC I:1.1/4 XIC B3:4/3 BST TON T4:19 0.01 100 0 NXB XIC T4:19/DN OTE B3:4/2 BND EOR
%   B3:0/12  AUTO_ENGAGED  "AUTO SYSTEM ENGAGED" %
%   I:1.1/4  PLANER_DECK_RUN_CONF  "Planer Infeed Deck Run Confirm" %
%   B3:4/3  AUTO_START_IF_DECK  "AUTO START PLANER INFEED DECK" %
%   T4:19  GRADE_AUTO_START  "GRADE DECK AUTO START DELAY" %
%   B3:4/2  AUTO_START_GRADE  "AUTO START GRADE DECK" %
% Rung: 13 %
SOR XIC B3:0/12 XIC I:1.1/12 XIC B3:4/4 XIC B3:0/9 BST TON T4:20 0.01 25 0 NXB XIC T4:20/DN OTE B3:4/3 BND EOR
%   B3:0/12  AUTO_ENGAGED  "AUTO SYSTEM ENGAGED" %
%   I:1.1/12  IF_ROLLS_2_RUN_CONF  "Infeed Rolls #2 Run Confirm" %
%   B3:4/4  AUTO_START_ROLLS  "Auto Start Infeed Rolls" %
%   B3:0/9  BOARD_REQUEST  "Board Request" %
%   T4:20  IF_DECK_START_DELAY  "PLANER INFEED DECK AUTO START DELAY" %
%   B3:4/3  AUTO_START_IF_DECK  "AUTO START PLANER INFEED DECK" %

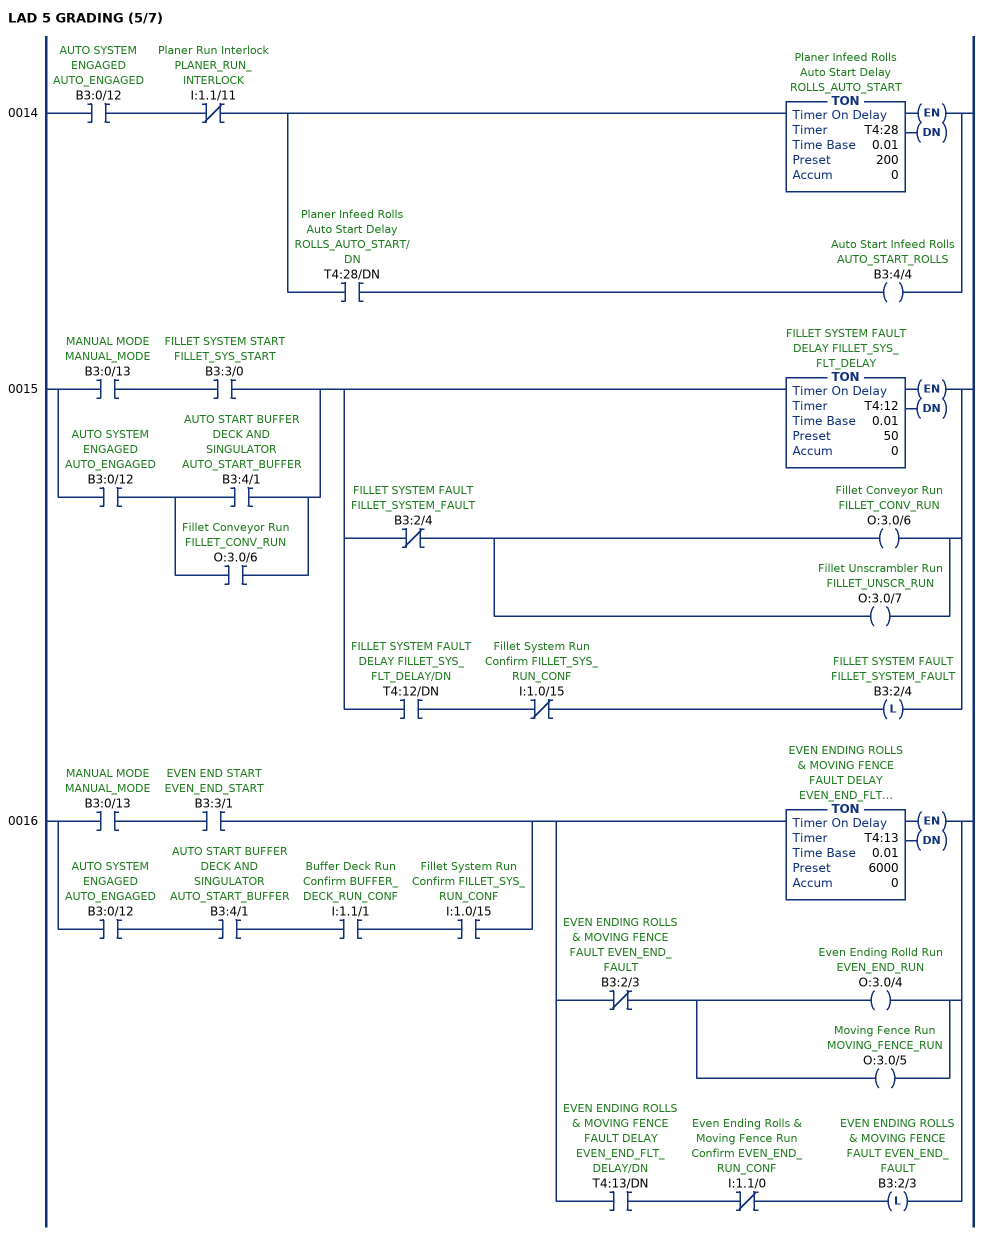
% Rung: 14 %
SOR XIC B3:0/12 XIO I:1.1/11 BST TON T4:28 0.01 200 0 NXB XIC T4:28/DN OTE B3:4/4 BND EOR
%   B3:0/12  AUTO_ENGAGED  "AUTO SYSTEM ENGAGED" %
%   I:1.1/11  PLANER_RUN_INTERLOCK  "Planer Run Interlock" %
%   T4:28  ROLLS_AUTO_START  "Planer Infeed Rolls Auto Start Delay" %
%   B3:4/4  AUTO_START_ROLLS  "Auto Start Infeed Rolls" %
% Rung: 15 %
SOR BST XIC B3:0/13 XIC B3:3/0 NXB XIC B3:0/12 BST XIC B3:4/1 NXB XIC O:3.0/6 BND BND BST TON T4:12 0.01 50 0 NXB XIO B3:2/4 BST OTE O:3.0/6 NXB OTE O:3.0/7 BND NXB XIC T4:12/DN XIO I:1.0/15 OTL B3:2/4 BND EOR
%   B3:0/13  MANUAL_MODE  "MANUAL MODE" %
%   B3:3/0  FILLET_SYS_START  "FILLET SYSTEM START" %
%   B3:0/12  AUTO_ENGAGED  "AUTO SYSTEM ENGAGED" %
%   B3:4/1  AUTO_START_BUFFER  "AUTO START BUFFER DECK AND SINGULATOR" %
%   O:3.0/6  FILLET_CONV_RUN  "Fillet Conveyor Run" %
%   T4:12  FILLET_SYS_FLT_DELAY  "FILLET SYSTEM FAULT DELAY" %
%   B3:2/4  FILLET_SYSTEM_FAULT  "FILLET SYSTEM FAULT" %
%   O:3.0/7  FILLET_UNSCR_RUN  "Fillet Unscrambler Run" %
%   I:1.0/15  FILLET_SYS_RUN_CONF  "Fillet System Run Confirm" %
% Rung: 16 %
SOR BST XIC B3:0/13 XIC B3:3/1 NXB XIC B3:0/12 XIC B3:4/1 XIC I:1.1/1 XIC I:1.0/15 BND BST TON T4:13 0.01 6000 0 NXB XIO B3:2/3 BST OTE O:3.0/4 NXB OTE O:3.0/5 BND NXB XIC T4:13/DN XIO I:1.1/0 OTL B3:2/3 BND EOR
%   B3:0/13  MANUAL_MODE  "MANUAL MODE" %
%   B3:3/1  EVEN_END_START  "EVEN END START" %
%   B3:0/12  AUTO_ENGAGED  "AUTO SYSTEM ENGAGED" %
%   B3:4/1  AUTO_START_BUFFER  "AUTO START BUFFER DECK AND SINGULATOR" %
%   I:1.1/1  BUFFER_DECK_RUN_CONF  "Buffer Deck Run Confirm" %
%   I:1.0/15  FILLET_SYS_RUN_CONF  "Fillet System Run Confirm" %
%   T4:13  EVEN_END_FLT_DELAY  "EVEN ENDING ROLLS & MOVING FENCE FAULT DELAY" %
%   B3:2/3  EVEN_END_FAULT  "EVEN ENDING ROLLS & MOVING FENCE FAULT" %
%   O:3.0/4  EVEN_END_RUN  "Even Ending Rolld Run" %
%   O:3.0/5  MOVING_FENCE_RUN  "Moving Fence Run" %
%   I:1.1/0  EVEN_END_RUN_CONF  "Even Ending Rolls & Moving Fence Run Confirm" %

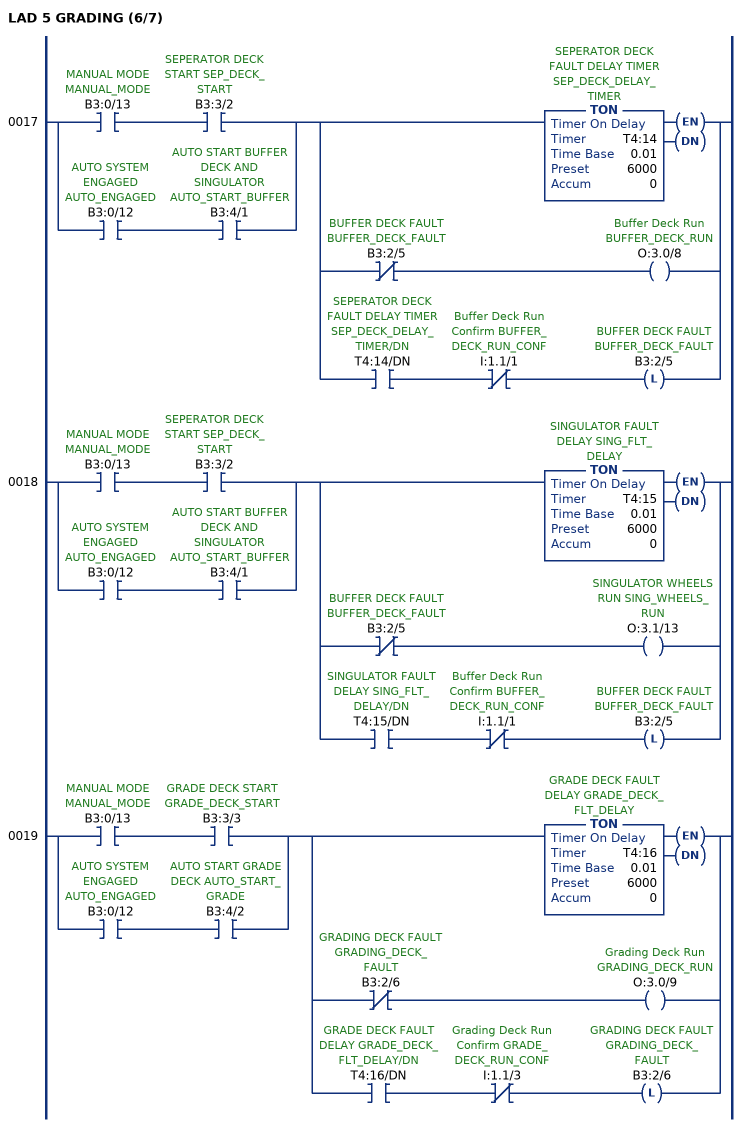
% Rung: 17 %
SOR BST XIC B3:0/13 XIC B3:3/2 NXB XIC B3:0/12 XIC B3:4/1 BND BST TON T4:14 0.01 6000 0 NXB XIO B3:2/5 OTE O:3.0/8 NXB XIC T4:14/DN XIO I:1.1/1 OTL B3:2/5 BND EOR
%   B3:0/13  MANUAL_MODE  "MANUAL MODE" %
%   B3:3/2  SEP_DECK_START  "SEPERATOR DECK START" %
%   B3:0/12  AUTO_ENGAGED  "AUTO SYSTEM ENGAGED" %
%   B3:4/1  AUTO_START_BUFFER  "AUTO START BUFFER DECK AND SINGULATOR" %
%   T4:14  SEP_DECK_DELAY_TIMER  "SEPERATOR DECK FAULT DELAY TIMER" %
%   B3:2/5  BUFFER_DECK_FAULT  "BUFFER DECK FAULT" %
%   O:3.0/8  BUFFER_DECK_RUN  "Buffer Deck Run" %
%   I:1.1/1  BUFFER_DECK_RUN_CONF  "Buffer Deck Run Confirm" %
% Rung: 18 %
SOR BST XIC B3:0/13 XIC B3:3/2 NXB XIC B3:0/12 XIC B3:4/1 BND BST TON T4:15 0.01 6000 0 NXB XIO B3:2/5 OTE O:3.1/13 NXB XIC T4:15/DN XIO I:1.1/1 OTL B3:2/5 BND EOR
%   B3:0/13  MANUAL_MODE  "MANUAL MODE" %
%   B3:3/2  SEP_DECK_START  "SEPERATOR DECK START" %
%   B3:0/12  AUTO_ENGAGED  "AUTO SYSTEM ENGAGED" %
%   B3:4/1  AUTO_START_BUFFER  "AUTO START BUFFER DECK AND SINGULATOR" %
%   T4:15  SING_FLT_DELAY  "SINGULATOR FAULT DELAY" %
%   B3:2/5  BUFFER_DECK_FAULT  "BUFFER DECK FAULT" %
%   O:3.1/13  SING_WHEELS_RUN  "SINGULATOR WHEELS RUN" %
%   I:1.1/1  BUFFER_DECK_RUN_CONF  "Buffer Deck Run Confirm" %
% Rung: 19 %
SOR BST XIC B3:0/13 XIC B3:3/3 NXB XIC B3:0/12 XIC B3:4/2 BND BST TON T4:16 0.01 6000 0 NXB XIO B3:2/6 OTE O:3.0/9 NXB XIC T4:16/DN XIO I:1.1/3 OTL B3:2/6 BND EOR
%   B3:0/13  MANUAL_MODE  "MANUAL MODE" %
%   B3:3/3  GRADE_DECK_START  "GRADE DECK START" %
%   B3:0/12  AUTO_ENGAGED  "AUTO SYSTEM ENGAGED" %
%   B3:4/2  AUTO_START_GRADE  "AUTO START GRADE DECK" %
%   T4:16  GRADE_DECK_FLT_DELAY  "GRADE DECK FAULT DELAY" %
%   B3:2/6  GRADING_DECK_FAULT  "GRADING DECK FAULT" %
%   O:3.0/9  GRADING_DECK_RUN  "Grading Deck Run" %
%   I:1.1/3  GRADE_DECK_RUN_CONF  "Grading Deck Run Confirm" %

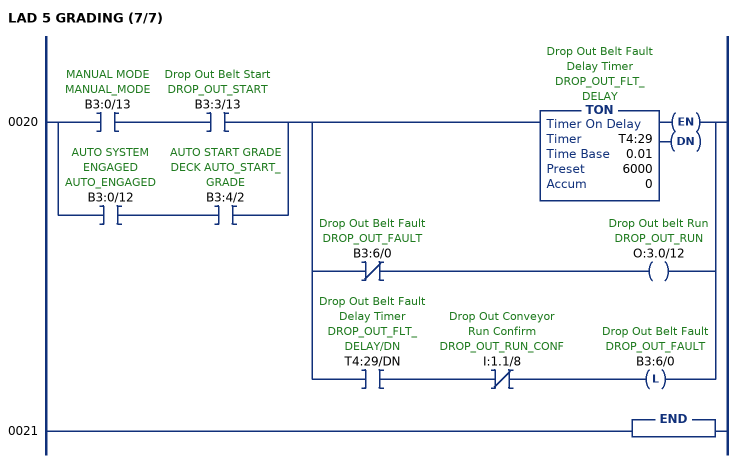
% Rung: 20 %
SOR BST XIC B3:0/13 XIC B3:3/13 NXB XIC B3:0/12 XIC B3:4/2 BND BST TON T4:29 0.01 6000 0 NXB XIO B3:6/0 OTE O:3.0/12 NXB XIC T4:29/DN XIO I:1.1/8 OTL B3:6/0 BND EOR
%   B3:0/13  MANUAL_MODE  "MANUAL MODE" %
%   B3:3/13  DROP_OUT_START  "Drop Out Belt Start" %
%   B3:0/12  AUTO_ENGAGED  "AUTO SYSTEM ENGAGED" %
%   B3:4/2  AUTO_START_GRADE  "AUTO START GRADE DECK" %
%   T4:29  DROP_OUT_FLT_DELAY  "Drop Out Belt Fault Delay Timer" %
%   B3:6/0  DROP_OUT_FAULT  "Drop Out Belt Fault" %
%   O:3.0/12  DROP_OUT_RUN  "Drop Out belt Run" %
%   I:1.1/8  DROP_OUT_RUN_CONF  "Drop Out Conveyor Run Confirm" %
% Rung: 21 %
SOR END EOR

LADDER 6 "PLANER IF"
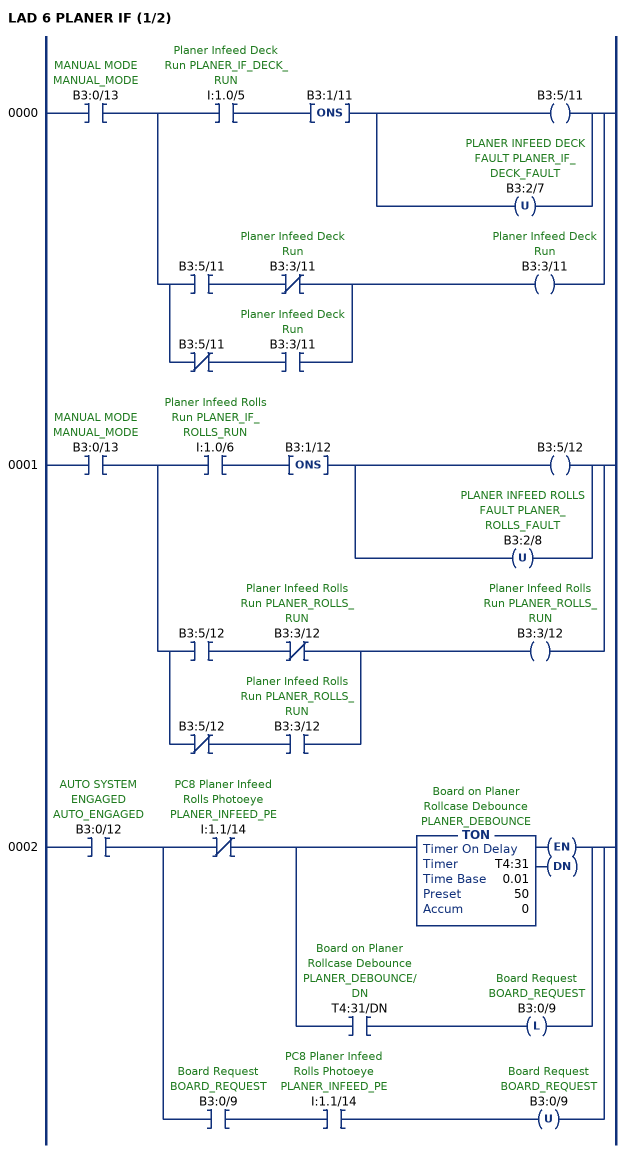
% Rung: 0 %
SOR XIC B3:0/13 BST XIC I:1.0/5 ONS B3:1/11 BST OTE B3:5/11 NXB OTU B3:2/7 BND NXB BST XIC B3:5/11 XIO B3:3/11 NXB XIO B3:5/11 XIC B3:3/11 BND OTE B3:3/11 BND EOR
%   B3:0/13  MANUAL_MODE  "MANUAL MODE" %
%   I:1.0/5  PLANER_IF_DECK_RUN  "Planer Infeed Deck Run" %
%   B3:2/7  PLANER_IF_DECK_FAULT  "PLANER INFEED DECK FAULT" %
%   B3:3/11  "Planer Infeed Deck Run" %
% Rung: 1 %
SOR XIC B3:0/13 BST XIC I:1.0/6 ONS B3:1/12 BST OTE B3:5/12 NXB OTU B3:2/8 BND NXB BST XIC B3:5/12 XIO B3:3/12 NXB XIO B3:5/12 XIC B3:3/12 BND OTE B3:3/12 BND EOR
%   B3:0/13  MANUAL_MODE  "MANUAL MODE" %
%   I:1.0/6  PLANER_IF_ROLLS_RUN  "Planer Infeed Rolls Run" %
%   B3:2/8  PLANER_ROLLS_FAULT  "PLANER INFEED ROLLS FAULT" %
%   B3:3/12  PLANER_ROLLS_RUN  "Planer Infeed Rolls Run" %
% Rung: 2 %
SOR XIC B3:0/12 BST XIO I:1.1/14 BST TON T4:31 0.01 50 0 NXB XIC T4:31/DN OTL B3:0/9 BND NXB XIC B3:0/9 XIC I:1.1/14 OTU B3:0/9 BND EOR
%   B3:0/12  AUTO_ENGAGED  "AUTO SYSTEM ENGAGED" %
%   I:1.1/14  PLANER_INFEED_PE  "PC8 Planer Infeed Rolls Photoeye" %
%   T4:31  PLANER_DEBOUNCE  "Board on Planer Rollcase Debounce" %
%   B3:0/9  BOARD_REQUEST  "Board Request" %

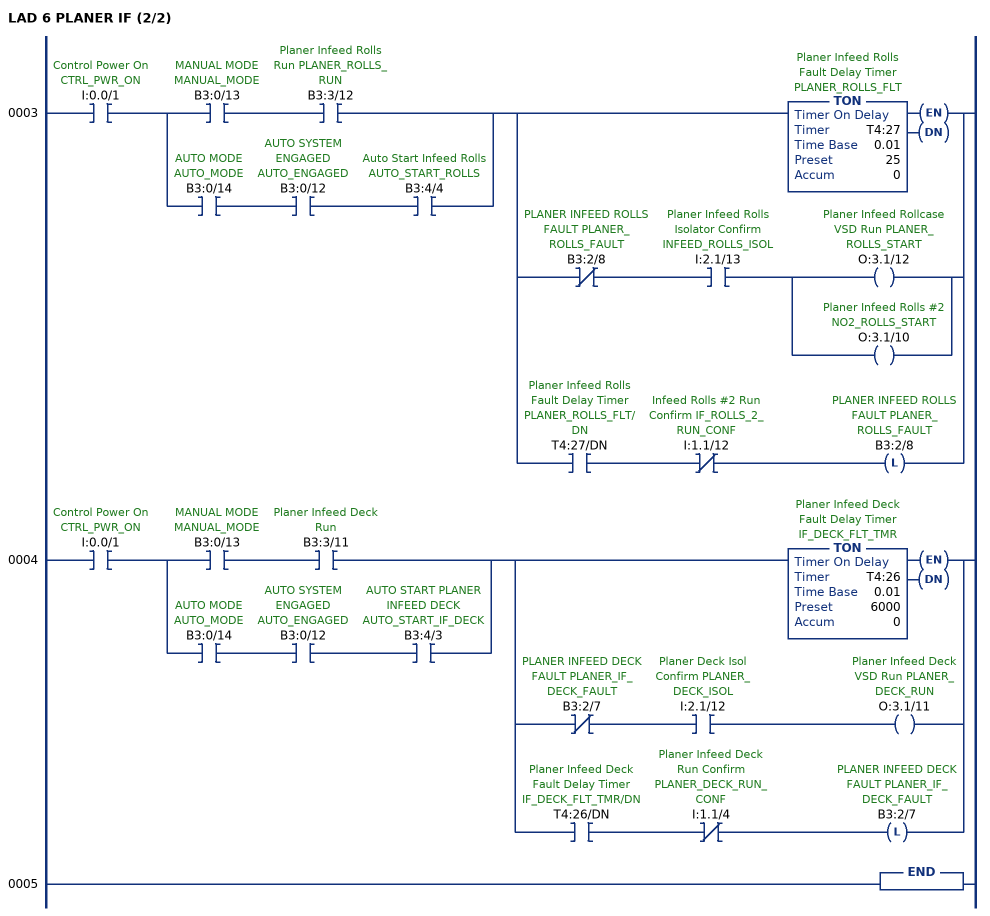
% Rung: 3 %
SOR XIC I:0.0/1 BST XIC B3:0/13 XIC B3:3/12 NXB XIC B3:0/14 XIC B3:0/12 XIC B3:4/4 BND BST TON T4:27 0.01 25 0 NXB XIO B3:2/8 XIC I:2.1/13 BST OTE O:3.1/12 NXB OTE O:3.1/10 BND NXB XIC T4:27/DN XIO I:1.1/12 OTL B3:2/8 BND EOR
%   I:0.0/1  CTRL_PWR_ON  "Control Power On" %
%   B3:0/13  MANUAL_MODE  "MANUAL MODE" %
%   B3:3/12  PLANER_ROLLS_RUN  "Planer Infeed Rolls Run" %
%   B3:0/14  AUTO_MODE  "AUTO MODE" %
%   B3:0/12  AUTO_ENGAGED  "AUTO SYSTEM ENGAGED" %
%   B3:4/4  AUTO_START_ROLLS  "Auto Start Infeed Rolls" %
%   T4:27  PLANER_ROLLS_FLT  "Planer Infeed Rolls Fault Delay Timer" %
%   B3:2/8  PLANER_ROLLS_FAULT  "PLANER INFEED ROLLS FAULT" %
%   I:2.1/13  INFEED_ROLLS_ISOL  "Planer Infeed Rolls Isolator Confirm" %
%   O:3.1/12  PLANER_ROLLS_START  "Planer Infeed Rollcase VSD Run" %
%   O:3.1/10  NO2_ROLLS_START  "Planer Infeed Rolls #2" %
%   I:1.1/12  IF_ROLLS_2_RUN_CONF  "Infeed Rolls #2 Run Confirm" %
% Rung: 4 %
SOR XIC I:0.0/1 BST XIC B3:0/13 XIC B3:3/11 NXB XIC B3:0/14 XIC B3:0/12 XIC B3:4/3 BND BST TON T4:26 0.01 6000 0 NXB XIO B3:2/7 XIC I:2.1/12 OTE O:3.1/11 NXB XIC T4:26/DN XIO I:1.1/4 OTL B3:2/7 BND EOR
%   I:0.0/1  CTRL_PWR_ON  "Control Power On" %
%   B3:0/13  MANUAL_MODE  "MANUAL MODE" %
%   B3:3/11  "Planer Infeed Deck Run" %
%   B3:0/14  AUTO_MODE  "AUTO MODE" %
%   B3:0/12  AUTO_ENGAGED  "AUTO SYSTEM ENGAGED" %
%   B3:4/3  AUTO_START_IF_DECK  "AUTO START PLANER INFEED DECK" %
%   T4:26  IF_DECK_FLT_TMR  "Planer Infeed Deck Fault Delay Timer" %
%   B3:2/7  PLANER_IF_DECK_FAULT  "PLANER INFEED DECK FAULT" %
%   I:2.1/12  PLANER_DECK_ISOL  "Planer Deck Isol Confirm" %
%   O:3.1/11  PLANER_DECK_RUN  "Planer Infeed Deck VSD Run" %
%   I:1.1/4  PLANER_DECK_RUN_CONF  "Planer Infeed Deck Run Confirm" %
% Rung: 5 %
SOR END EOR

LADDER 7 "PLANER OF"
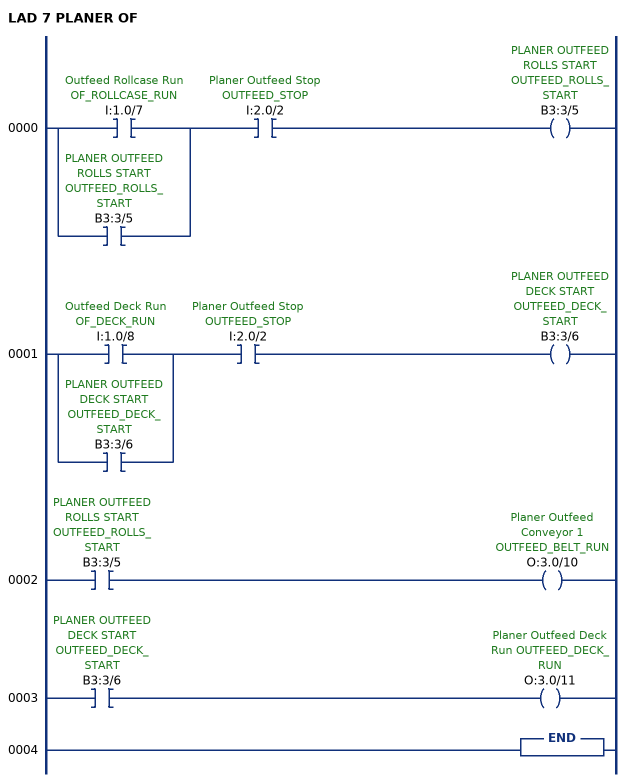
% Rung: 0 %
SOR BST XIC I:1.0/7 NXB XIC B3:3/5 BND XIC I:2.0/2 OTE B3:3/5 EOR
%   I:1.0/7  OF_ROLLCASE_RUN  "Outfeed Rollcase Run" %
%   B3:3/5  OUTFEED_ROLLS_START  "PLANER OUTFEED ROLLS START" %
%   I:2.0/2  OUTFEED_STOP  "Planer Outfeed Stop" %
% Rung: 1 %
SOR BST XIC I:1.0/8 NXB XIC B3:3/6 BND XIC I:2.0/2 OTE B3:3/6 EOR
%   I:1.0/8  OF_DECK_RUN  "Outfeed Deck Run" %
%   B3:3/6  OUTFEED_DECK_START  "PLANER OUTFEED DECK START" %
%   I:2.0/2  OUTFEED_STOP  "Planer Outfeed Stop" %
% Rung: 2 %
SOR XIC B3:3/5 OTE O:3.0/10 EOR
%   B3:3/5  OUTFEED_ROLLS_START  "PLANER OUTFEED ROLLS START" %
%   O:3.0/10  OUTFEED_BELT_RUN  "Planer Outfeed Conveyor 1" %
% Rung: 3 %
SOR XIC B3:3/6 OTE O:3.0/11 EOR
%   B3:3/6  OUTFEED_DECK_START  "PLANER OUTFEED DECK START" %
%   O:3.0/11  OUTFEED_DECK_RUN  "Planer Outfeed Deck Run" %
% Rung: 4 %
SOR END EOR

LADDER 8 "MR CONVS"
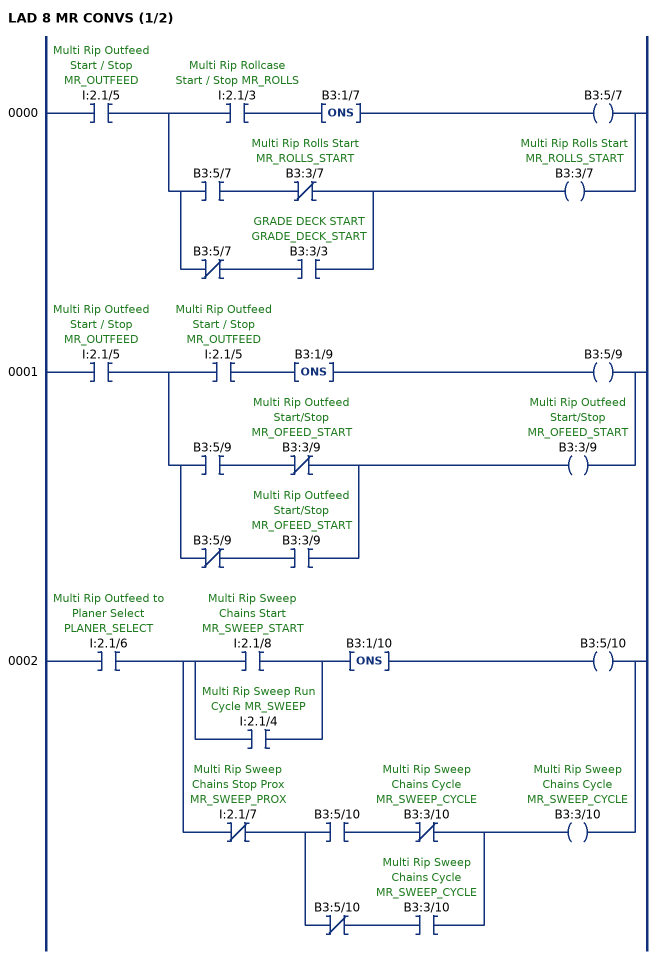
% Rung: 0 %
SOR XIC I:2.1/5 BST XIC I:2.1/3 ONS B3:1/7 OTE B3:5/7 NXB BST XIC B3:5/7 XIO B3:3/7 NXB XIO B3:5/7 XIC B3:3/3 BND OTE B3:3/7 BND EOR
%   I:2.1/5  MR_OUTFEED  "Multi Rip Outfeed Start / Stop" %
%   I:2.1/3  MR_ROLLS  "Multi Rip Rollcase Start / Stop" %
%   B3:3/7  MR_ROLLS_START  "Multi Rip Rolls Start" %
%   B3:3/3  GRADE_DECK_START  "GRADE DECK START" %
% Rung: 1 %
SOR XIC I:2.1/5 BST XIC I:2.1/5 ONS B3:1/9 OTE B3:5/9 NXB BST XIC B3:5/9 XIO B3:3/9 NXB XIO B3:5/9 XIC B3:3/9 BND OTE B3:3/9 BND EOR
%   I:2.1/5  MR_OUTFEED  "Multi Rip Outfeed Start / Stop" %
%   B3:3/9  MR_OFEED_START  "Multi Rip Outfeed Start/Stop" %
% Rung: 2 %
SOR XIC I:2.1/6 BST BST XIC I:2.1/8 NXB XIC I:2.1/4 BND ONS B3:1/10 OTE B3:5/10 NXB XIO I:2.1/7 BST XIC B3:5/10 XIO B3:3/10 NXB XIO B3:5/10 XIC B3:3/10 BND OTE B3:3/10 BND EOR
%   I:2.1/6  PLANER_SELECT  "Multi Rip Outfeed to Planer Select" %
%   I:2.1/8  MR_SWEEP_START  "Multi Rip Sweep Chains Start" %
%   I:2.1/4  MR_SWEEP  "Multi Rip Sweep Run Cycle" %
%   I:2.1/7  MR_SWEEP_PROX  "Multi Rip Sweep Chains Stop Prox" %
%   B3:3/10  MR_SWEEP_CYCLE  "Multi Rip Sweep Chains Cycle" %

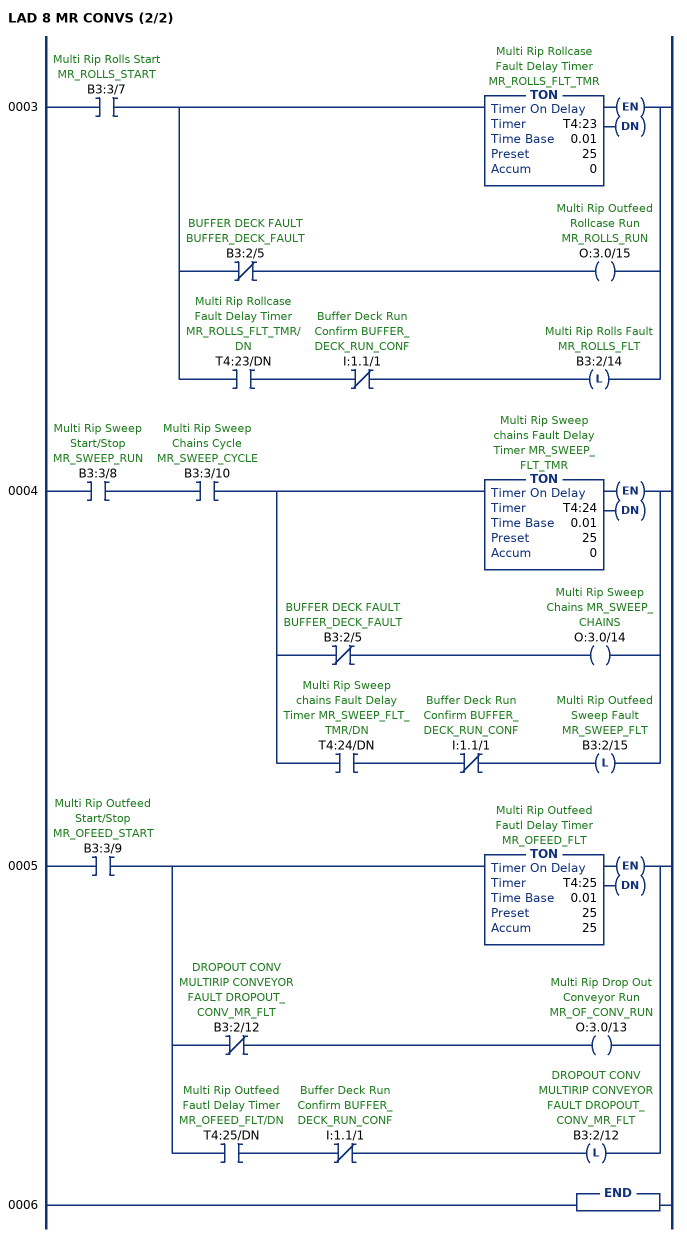
% Rung: 3 %
SOR XIC B3:3/7 BST TON T4:23 0.01 25 0 NXB XIO B3:2/5 OTE O:3.0/15 NXB XIC T4:23/DN XIO I:1.1/1 OTL B3:2/14 BND EOR
%   B3:3/7  MR_ROLLS_START  "Multi Rip Rolls Start" %
%   T4:23  MR_ROLLS_FLT_TMR  "Multi Rip Rollcase Fault Delay Timer" %
%   B3:2/5  BUFFER_DECK_FAULT  "BUFFER DECK FAULT" %
%   O:3.0/15  MR_ROLLS_RUN  "Multi Rip Outfeed Rollcase Run" %
%   I:1.1/1  BUFFER_DECK_RUN_CONF  "Buffer Deck Run Confirm" %
%   B3:2/14  MR_ROLLS_FLT  "Multi Rip Rolls Fault" %
% Rung: 4 %
SOR XIC B3:3/8 XIC B3:3/10 BST TON T4:24 0.01 25 0 NXB XIO B3:2/5 OTE O:3.0/14 NXB XIC T4:24/DN XIO I:1.1/1 OTL B3:2/15 BND EOR
%   B3:3/8  MR_SWEEP_RUN  "Multi Rip Sweep Start/Stop" %
%   B3:3/10  MR_SWEEP_CYCLE  "Multi Rip Sweep Chains Cycle" %
%   T4:24  MR_SWEEP_FLT_TMR  "Multi Rip Sweep chains Fault Delay Timer" %
%   B3:2/5  BUFFER_DECK_FAULT  "BUFFER DECK FAULT" %
%   O:3.0/14  MR_SWEEP_CHAINS  "Multi Rip Sweep Chains" %
%   I:1.1/1  BUFFER_DECK_RUN_CONF  "Buffer Deck Run Confirm" %
%   B3:2/15  MR_SWEEP_FLT  "Multi Rip Outfeed Sweep Fault" %
% Rung: 5 %
SOR XIC B3:3/9 BST TON T4:25 0.01 25 25 NXB XIO B3:2/12 OTE O:3.0/13 NXB XIC T4:25/DN XIO I:1.1/1 OTL B3:2/12 BND EOR
%   B3:3/9  MR_OFEED_START  "Multi Rip Outfeed Start/Stop" %
%   T4:25  MR_OFEED_FLT  "Multi Rip Outfeed Fautl Delay Timer" %
%   B3:2/12  DROPOUT_CONV_MR_FLT  "DROPOUT CONV MULTIRIP CONVEYOR FAULT" %
%   O:3.0/13  MR_OF_CONV_RUN  "Multi Rip Drop Out Conveyor Run" %
%   I:1.1/1  BUFFER_DECK_RUN_CONF  "Buffer Deck Run Confirm" %
% Rung: 6 %
SOR END EOR

LADDER 9 "CYCLONE"
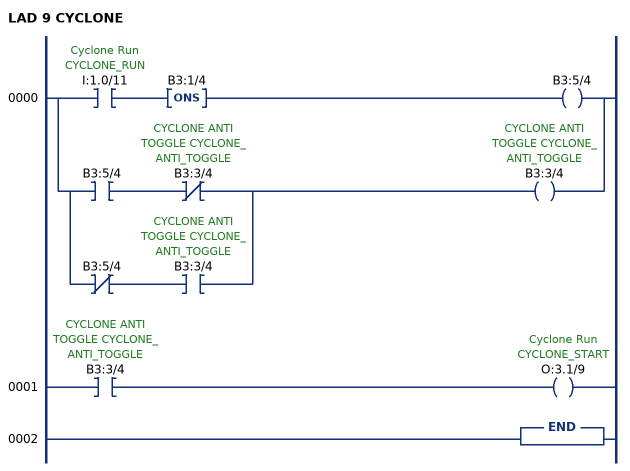
% Rung: 0 %
SOR BST XIC I:1.0/11 ONS B3:1/4 OTE B3:5/4 NXB BST XIC B3:5/4 XIO B3:3/4 NXB XIO B3:5/4 XIC B3:3/4 BND OTE B3:3/4 BND EOR
%   I:1.0/11  CYCLONE_RUN  "Cyclone Run" %
%   B3:3/4  CYCLONE_ANTI_TOGGLE  "CYCLONE ANTI TOGGLE" %
% Rung: 1 %
SOR XIC B3:3/4 OTE O:3.1/9 EOR
%   B3:3/4  CYCLONE_ANTI_TOGGLE  "CYCLONE ANTI TOGGLE" %
%   O:3.1/9  CYCLONE_START  "Cyclone Run" %
% Rung: 2 %
SOR END EOR

LADDER 10 "INDICATION"
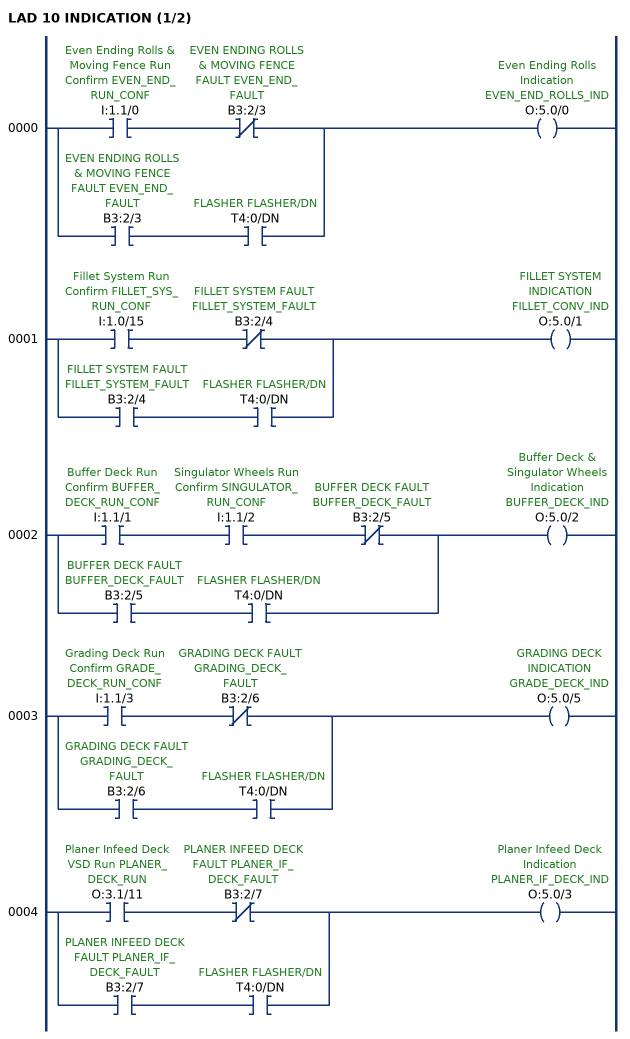
% Rung: 0 %
SOR BST XIC I:1.1/0 XIO B3:2/3 NXB XIC B3:2/3 XIC T4:0/DN BND OTE O:5.0/0 EOR
%   I:1.1/0  EVEN_END_RUN_CONF  "Even Ending Rolls & Moving Fence Run Confirm" %
%   B3:2/3  EVEN_END_FAULT  "EVEN ENDING ROLLS & MOVING FENCE FAULT" %
%   T4:0  FLASHER  "FLASHER" %
%   O:5.0/0  EVEN_END_ROLLS_IND  "Even Ending Rolls Indication" %
% Rung: 1 %
SOR BST XIC I:1.0/15 XIO B3:2/4 NXB XIC B3:2/4 XIC T4:0/DN BND OTE O:5.0/1 EOR
%   I:1.0/15  FILLET_SYS_RUN_CONF  "Fillet System Run Confirm" %
%   B3:2/4  FILLET_SYSTEM_FAULT  "FILLET SYSTEM FAULT" %
%   T4:0  FLASHER  "FLASHER" %
%   O:5.0/1  FILLET_CONV_IND  "FILLET SYSTEM INDICATION" %
% Rung: 2 %
SOR BST XIC I:1.1/1 XIC I:1.1/2 XIO B3:2/5 NXB XIC B3:2/5 XIC T4:0/DN BND OTE O:5.0/2 EOR
%   I:1.1/1  BUFFER_DECK_RUN_CONF  "Buffer Deck Run Confirm" %
%   I:1.1/2  SINGULATOR_RUN_CONF  "Singulator Wheels Run Confirm" %
%   B3:2/5  BUFFER_DECK_FAULT  "BUFFER DECK FAULT" %
%   T4:0  FLASHER  "FLASHER" %
%   O:5.0/2  BUFFER_DECK_IND  "Buffer Deck & Singulator Wheels Indication" %
% Rung: 3 %
SOR BST XIC I:1.1/3 XIO B3:2/6 NXB XIC B3:2/6 XIC T4:0/DN BND OTE O:5.0/5 EOR
%   I:1.1/3  GRADE_DECK_RUN_CONF  "Grading Deck Run Confirm" %
%   B3:2/6  GRADING_DECK_FAULT  "GRADING DECK FAULT" %
%   T4:0  FLASHER  "FLASHER" %
%   O:5.0/5  GRADE_DECK_IND  "GRADING DECK INDICATION" %
% Rung: 4 %
SOR BST XIC O:3.1/11 XIO B3:2/7 NXB XIC B3:2/7 XIC T4:0/DN BND OTE O:5.0/3 EOR
%   O:3.1/11  PLANER_DECK_RUN  "Planer Infeed Deck VSD Run" %
%   B3:2/7  PLANER_IF_DECK_FAULT  "PLANER INFEED DECK FAULT" %
%   T4:0  FLASHER  "FLASHER" %
%   O:5.0/3  PLANER_IF_DECK_IND  "Planer Infeed Deck Indication" %

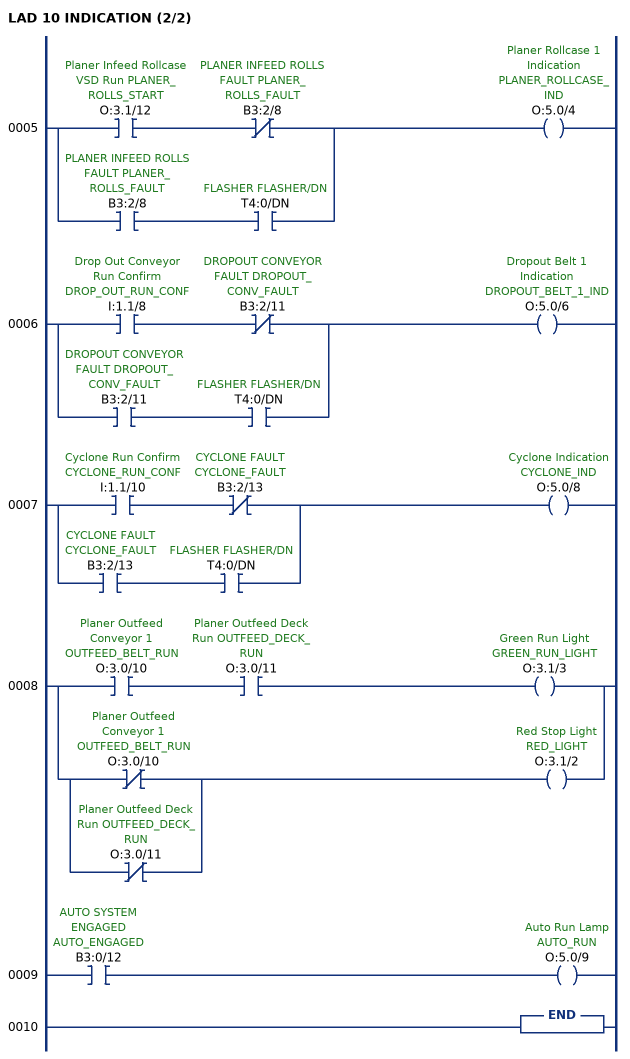
% Rung: 5 %
SOR BST XIC O:3.1/12 XIO B3:2/8 NXB XIC B3:2/8 XIC T4:0/DN BND OTE O:5.0/4 EOR
%   O:3.1/12  PLANER_ROLLS_START  "Planer Infeed Rollcase VSD Run" %
%   B3:2/8  PLANER_ROLLS_FAULT  "PLANER INFEED ROLLS FAULT" %
%   T4:0  FLASHER  "FLASHER" %
%   O:5.0/4  PLANER_ROLLCASE_IND  "Planer Rollcase 1 Indication" %
% Rung: 6 %
SOR BST XIC I:1.1/8 XIO B3:2/11 NXB XIC B3:2/11 XIC T4:0/DN BND OTE O:5.0/6 EOR
%   I:1.1/8  DROP_OUT_RUN_CONF  "Drop Out Conveyor Run Confirm" %
%   B3:2/11  DROPOUT_CONV_FAULT  "DROPOUT CONVEYOR FAULT" %
%   T4:0  FLASHER  "FLASHER" %
%   O:5.0/6  DROPOUT_BELT_1_IND  "Dropout Belt 1 Indication" %
% Rung: 7 %
SOR BST XIC I:1.1/10 XIO B3:2/13 NXB XIC B3:2/13 XIC T4:0/DN BND OTE O:5.0/8 EOR
%   I:1.1/10  CYCLONE_RUN_CONF  "Cyclone Run Confirm" %
%   B3:2/13  CYCLONE_FAULT  "CYCLONE FAULT" %
%   T4:0  FLASHER  "FLASHER" %
%   O:5.0/8  CYCLONE_IND  "Cyclone Indication" %
% Rung: 8 %
SOR BST XIC O:3.0/10 XIC O:3.0/11 OTE O:3.1/3 NXB BST XIO O:3.0/10 NXB XIO O:3.0/11 BND OTE O:3.1/2 BND EOR
%   O:3.0/10  OUTFEED_BELT_RUN  "Planer Outfeed Conveyor 1" %
%   O:3.0/11  OUTFEED_DECK_RUN  "Planer Outfeed Deck Run" %
%   O:3.1/3  GREEN_RUN_LIGHT  "Green Run Light" %
%   O:3.1/2  RED_LIGHT  "Red Stop Light" %
% Rung: 9 %
SOR XIC B3:0/12 OTE O:5.0/9 EOR
%   B3:0/12  AUTO_ENGAGED  "AUTO SYSTEM ENGAGED" %
%   O:5.0/9  AUTO_RUN  "Auto Run Lamp" %
% Rung: 10 %
SOR END EOR

OTHER DOCUMENTED ADDRESSES
  B3:2/2  "TILT HOIST FAULT"
  B3:2/9  PLANER_OF_ROLLS_FLT  "PLANER OUTFEED ROLLS FLT"
  B3:2/10  PLANER_OF_DECK_FAULT  "PLANER OUTFEED DECK FAULT"
  I:0.0/3  SEMI_AUTO  "Semi Auto Mode"
  I:1.0/10  DROP_OUT_MR_CONV_RUN  "Drop Out Conveyor From Multi Rip Run"
  I:1.0/14  HOIST_RUN_CONF  "Tilt Hoist Run Confirm"
  I:1.1/5  IF_ROLLS_RUN_CONF  "Planer Infeed Rolls Run Confirm"
  I:1.1/6  OF_ROLLS_RUN_CONF  "Outfeed Rolls Run Confirm"
  I:1.1/7  OF_DECK_RUN_CONF  "Outfeed Deck Run Confirm"
  I:1.1/9  MR_CONV_RUN_CONF  "Drop Out Conveyor to Multi Rip Run Confirm"
  I:2.0/12  HOIST_ISOLATOR  "Tilt Hoist ISolator COnfirm"
  I:2.0/15  WHEELS_ISOL_CONFIRM  "Singulator Wheels Isolator Confirm"
  I:2.1/0  HOIST_VSD_FAULT  "Tilt Hoist VSD Fault"
  I:2.1/9  OUTFEED_ESTOP  "Outfeed EStop"
  I:2.1/10  MR_ROLLS_RUN_CONF  "Multi Rip Outfeed Rollcase Run Confirm"
  I:2.1/11  MR_SWEEP_RUN_CONF  "Multi Rip Sweep Chains Run Confirm"
  O:4.0/7  DROPOUT_BELT_MR_IND  "Dropout Belt Multirip Indication"
  T4:8  HOIST_UP_FLT_DELAY  "TILT HOIST UP FAULT DELAY"
  T4:10  HOIST_DOWN_FLT_DELAY  "TILT HOIST DOWN FAULT DELAY"
  T4:21  OUTFEED_ROLLS_DELAY  "PLANER OUTFEED ROLLS FAULT DELAY TIMER"
  T4:22  OUTFEED_DECK_DELAY  "PLANER OUTFEED DECK FAULT DELAY TIMER"

REVISION NOTES
  0: Onsite Programming 13-1-07
  1: 15-1-07 Final Commissioning and Semi Auto Mode Installed

DATA TABLE (non-zero values as saved)
DATA B3
% B3:0 % 0X2000 0X8200 0X1000 0X0300 0X0000 0X0000 0X0000 0X0000 0X0000 0X0000
DATA T4
% .PRE .ACC %
% T4:0 % 50 50
% T4:1 % 50 46
% T4:2 % 10 0
% T4:3 % 6000 0
% T4:4 % 6000 0
% T4:5 % 25 0
% T4:6 % 500 500
% T4:7 % 50 0
% T4:8 % 6000 0
% T4:9 % 1000 0
% T4:10 % 6000 0
% T4:11 % 50 0
% T4:12 % 50 0
% T4:13 % 6000 0
% T4:14 % 6000 0
% T4:15 % 6000 0
% T4:16 % 6000 0
% T4:17 % 100 0
% T4:18 % 100 0
% T4:19 % 100 0
% T4:20 % 25 0
% T4:21 % 25 0
% T4:22 % 25 0
% T4:23 % 25 0
% T4:24 % 25 0
% T4:25 % 25 25
% T4:26 % 6000 0
% T4:27 % 25 0
% T4:28 % 200 0
% T4:29 % 6000 0
% T4:30 % 500 0
% T4:31 % 50 0
% T4:32 % 500 0
% T4:33 % 600 600
